(* IEC 61131-3 sources: UniTest/iecUniTest_br/iecUniTest, 121 files *)

(* ---- iecUniTest.typ ---- *)
TYPE
    utTestCase :    STRUCT
        id : UINT; (*Identifier of the test*)
        desc : ARRAY[0..4] OF STRING[255]; (*Description of the test case*)
        state : utTestCaseStates; (*State of the test*)
        msg : STRING[255]; (*Result of the test*)
    END_STRUCT;
    utTestCaseStates :
    (
        ut_SETUP := 0, (**)
        ut_RUNNING := 1, (**)
        ut_PASSED := 2, (**)
        ut_FAILED := 3, (**)
    )
    utTestCaseSummary :    STRUCT
        Id : UINT; (*Id of the test object. Must be unique number*)
        Name : STRING[250]; (*Name of the test object*)
        TotalTests : UINT; (*Total number of tests existing*)
        TestsPassed : UINT; (*Number of tests passed*)
        TestsFailed : UINT; (*Number of tests failed*)
        PassRate : REAL; (*Pass rate % of the tests*)
        TestsRunning : BOOL; (*One or more tests are running*)
        Error : utErrors; (*Error code if error occured*)
    END_STRUCT;
    utErrors :
    (
        ut_NO_ERROR := 0, (**)
        ut_NO_TEST_CASES_DEFINED := 100, (**)
    )
END_TYPE

(* ---- assertArrayEqual_BOOL.st ---- *)
FUNCTION assertArrayEqual_BOOL
    (*https://github.com/tkucic/iecUniTest/blob/main/docs/docs/ns/iecUniTest/fc/assertArrayEqual_BOOL.md*)
    vStop := (size / SIZEOF(act^[0])) - 1;

    FOR i:=0 TO vStop DO
    	pt1 := ADR(act^[i]);
    	pt2 := ADR(xp^[i]);
    	IF pt1^ <> pt2^ THEN
    		assertArrayEqual_BOOL := FALSE;
    		RETURN;
    	END_IF
    END_FOR
    (*If we reach here, all elements are equal*)
    assertArrayEqual_BOOL := TRUE;
    RETURN;

END_FUNCTION

(* ---- assertArrayEqual_BYTE.st ---- *)
FUNCTION assertArrayEqual_BYTE
    (*https://github.com/tkucic/iecUniTest/blob/main/docs/docs/ns/iecUniTest/fc/assertArrayEqual_BYTE.md*)
    vStop := (size / SIZEOF(act[0])) - 1;

    FOR i:=0 TO vStop DO
    	pt1 ACCESS ADR(act[i]);
    	pt2 ACCESS ADR(xp[i]);
    	IF pt1 <> pt2 THEN
    		assertArrayEqual_BYTE := FALSE;
    		RETURN;
    	END_IF
    END_FOR
    (*If we reach here, all elements are equal*)
    assertArrayEqual_BYTE := TRUE;
    RETURN;

END_FUNCTION

(* ---- assertArrayEqual_DATE.st ---- *)
FUNCTION assertArrayEqual_DATE
    (*https://github.com/tkucic/iecUniTest/blob/main/docs/docs/ns/iecUniTest/fc/assertArrayEqual_DATE.md*)
    vStop := (size / SIZEOF(act[0])) - 1;

    FOR i:=0 TO vStop DO
    	pt1 ACCESS ADR(act[i]);
    	pt2 ACCESS ADR(xp[i]);
    	IF pt1 <> pt2 THEN
    		assertArrayEqual_DATE := FALSE;
    		RETURN;
    	END_IF
    END_FOR
    (*If we reach here, all elements are equal*)
    assertArrayEqual_DATE := TRUE;
    RETURN;

END_FUNCTION

(* ---- assertArrayEqual_DATE_AND_TIME.st ---- *)
FUNCTION assertArrayEqual_DATE_AND_TIME
    (*https://github.com/tkucic/iecUniTest/blob/main/docs/docs/ns/iecUniTest/fc/assertArrayEqual_DATE_AND_TIME.md*)
    vStop := (size / SIZEOF(act[0])) - 1;

    FOR i:=0 TO vStop DO
    	pt1 ACCESS ADR(act[i]);
    	pt2 ACCESS ADR(xp[i]);
    	IF pt1 <> pt2 THEN
    		assertArrayEqual_DATE_AND_TIME := FALSE;
    		RETURN;
    	END_IF
    END_FOR
    (*If we reach here, all elements are equal*)
    assertArrayEqual_DATE_AND_TIME := TRUE;
    RETURN;

END_FUNCTION

(* ---- assertArrayEqual_DINT.st ---- *)
FUNCTION assertArrayEqual_DINT
    (*https://github.com/tkucic/iecUniTest/blob/main/docs/docs/ns/iecUniTest/fc/assertArrayEqual_DINT.md*)
    vStop := (size / SIZEOF(act[0])) - 1;

    FOR i:=0 TO vStop DO
    	pt1 ACCESS ADR(act[i]);
    	pt2 ACCESS ADR(xp[i]);
    	IF pt1 <> pt2 THEN
    		assertArrayEqual_DINT := FALSE;
    		RETURN;
    	END_IF
    END_FOR
    (*If we reach here, all elements are equal*)
    assertArrayEqual_DINT := TRUE;
    RETURN;

END_FUNCTION

(* ---- assertArrayEqual_DWORD.st ---- *)
FUNCTION assertArrayEqual_DWORD
    (*https://github.com/tkucic/iecUniTest/blob/main/docs/docs/ns/iecUniTest/fc/assertArrayEqual_DWORD.md*)
    vStop := (size / SIZEOF(act[0])) - 1;

    FOR i:=0 TO vStop DO
    	pt1 ACCESS ADR(act[i]);
    	pt2 ACCESS ADR(xp[i]);
    	IF pt1 <> pt2 THEN
    		assertArrayEqual_DWORD := FALSE;
    		RETURN;
    	END_IF
    END_FOR
    (*If we reach here, all elements are equal*)
    assertArrayEqual_DWORD := TRUE;
    RETURN;

END_FUNCTION

(* ---- assertArrayEqual_INT.st ---- *)
FUNCTION assertArrayEqual_INT
    (*https://github.com/tkucic/iecUniTest/blob/main/docs/docs/ns/iecUniTest/fc/assertArrayEqual_INT.md*)
    vStop := (size / SIZEOF(act[0])) - 1;

    FOR i:=0 TO vStop DO
    	pt1 ACCESS ADR(act[i]);
    	pt2 ACCESS ADR(xp[i]);
    	IF pt1 <> pt2 THEN
    		assertArrayEqual_INT := FALSE;
    		RETURN;
    	END_IF
    END_FOR
    (*If we reach here, all elements are equal*)
    assertArrayEqual_INT := TRUE;
    RETURN;

END_FUNCTION

(* ---- assertArrayEqual_LREAL.st ---- *)
FUNCTION assertArrayEqual_LREAL
    (*https://github.com/tkucic/iecUniTest/blob/main/docs/docs/ns/iecUniTest/fc/assertArrayEqual_LREAL.md*)
    vStop := (size / SIZEOF(act^[0])) - 1;

    FOR i:=0 TO vStop DO
    	pt1 := ADR(act^[i]);
    	pt2 := ADR(xp^[i]);
    	IF pt1^ <> pt2^ THEN
    		assertArrayEqual_LREAL := FALSE;
    		RETURN;
    	END_IF
    END_FOR
    (*If we reach here, all elements are equal*)
    assertArrayEqual_LREAL := TRUE;
    RETURN;

END_FUNCTION

(* ---- assertArrayEqual_REAL.st ---- *)
FUNCTION assertArrayEqual_REAL
    (*https://github.com/tkucic/iecUniTest/blob/main/docs/docs/ns/iecUniTest/fc/assertArrayEqual_REAL.md*)
    vStop := (size / SIZEOF(act^[0])) - 1;

    FOR i:=0 TO vStop DO
    	pt1 := ADR(act^[i]);
    	pt2 := ADR(xp^[i]);
    	IF pt1^ <> pt2^ THEN
    		assertArrayEqual_REAL := FALSE;
    		RETURN;
    	END_IF
    END_FOR
    (*If we reach here, all elements are equal*)
    assertArrayEqual_REAL := TRUE;
    RETURN;

END_FUNCTION

(* ---- assertArrayEqual_SINT.st ---- *)
FUNCTION assertArrayEqual_SINT
    (*https://github.com/tkucic/iecUniTest/blob/main/docs/docs/ns/iecUniTest/fc/assertArrayEqual_SINT.md*)
    vStop := (size / SIZEOF(act[0])) - 1;

    FOR i:=0 TO vStop DO
    	pt1 ACCESS ADR(act[i]);
    	pt2 ACCESS ADR(xp[i]);
    	IF pt1 <> pt2 THEN
    		assertArrayEqual_SINT := FALSE;
    		RETURN;
    	END_IF
    END_FOR
    (*If we reach here, all elements are equal*)
    assertArrayEqual_SINT := TRUE;
    RETURN;

END_FUNCTION

(* ---- assertArrayEqual_STRING.st ---- *)
FUNCTION assertArrayEqual_STRING
    (*https://github.com/tkucic/iecUniTest/blob/main/docs/docs/ns/iecUniTest/fc/assertArrayEqual_STRING.md*)
    vStop := (size / SIZEOF(act[0])) - 1;

    FOR i:=0 TO vStop DO
    	pt1 ACCESS ADR(act[i]);
    	pt2 ACCESS ADR(xp[i]);
    	IF pt1 <> pt2 THEN
    		assertArrayEqual_STRING := FALSE;
    		RETURN;
    	END_IF
    END_FOR
    (*If we reach here, all elements are equal*)
    assertArrayEqual_STRING := TRUE;
    RETURN;

END_FUNCTION

(* ---- assertArrayEqual_TIME.st ---- *)
FUNCTION assertArrayEqual_TIME
    (*https://github.com/tkucic/iecUniTest/blob/main/docs/docs/ns/iecUniTest/fc/assertArrayEqual_TIME.md*)
    vStop := (size / SIZEOF(act^[0])) - 1;

    FOR i:=0 TO vStop DO
    	pt1 := ADR(act^[i]);
    	pt2 := ADR(xp^[i]);
    	IF pt1^ <> pt2^ THEN
    		assertArrayEqual_TIME := FALSE;
    		RETURN;
    	END_IF
    END_FOR
    (*If we reach here, all elements are equal*)
    assertArrayEqual_TIME := TRUE;
    RETURN;

END_FUNCTION

(* ---- assertArrayEqual_TIME_OF_DAY.st ---- *)
FUNCTION assertArrayEqual_TIME_OF_DAY
    (*https://github.com/tkucic/iecUniTest/blob/main/docs/docs/ns/iecUniTest/fc/assertArrayEqual_TIME_OF_DAY.md*)
    vStop := (size / SIZEOF(act^[0])) - 1;

    FOR i:=0 TO vStop DO
    	pt1 := ADR(act^[i]);
    	pt2 := ADR(xp^[i]);
    	IF pt1^ <> pt2^ THEN
    		assertArrayEqual_TIME_OF_DAY := FALSE;
    		RETURN;
    	END_IF
    END_FOR
    (*If we reach here, all elements are equal*)
    assertArrayEqual_TIME_OF_DAY := TRUE;
    RETURN;

END_FUNCTION

(* ---- assertArrayEqual_UDINT.st ---- *)
FUNCTION assertArrayEqual_UDINT
    (*https://github.com/tkucic/iecUniTest/blob/main/docs/docs/ns/iecUniTest/fc/assertArrayEqual_UDINT.md*)
    vStop := (size / SIZEOF(act[0])) - 1;

    FOR i:=0 TO vStop DO
    	pt1 ACCESS ADR(act[i]);
    	pt2 ACCESS ADR(xp[i]);
    	IF pt1 <> pt2 THEN
    		assertArrayEqual_UDINT := FALSE;
    		RETURN;
    	END_IF
    END_FOR
    (*If we reach here, all elements are equal*)
    assertArrayEqual_UDINT := TRUE;
    RETURN;

END_FUNCTION

(* ---- assertArrayEqual_UINT.st ---- *)
FUNCTION assertArrayEqual_UINT
    (*https://github.com/tkucic/iecUniTest/blob/main/docs/docs/ns/iecUniTest/fc/assertArrayEqual_UINT.md*)
    vStop := (size / SIZEOF(act^[0])) - 1;

    FOR i:=0 TO vStop DO
    	pt1 := ADR(act^[i]);
    	pt2 := ADR(xp^[i]);
    	IF pt1^ <> pt2^ THEN
    		assertArrayEqual_UINT := FALSE;
    		RETURN;
    	END_IF
    END_FOR
    (*If we reach here, all elements are equal*)
    assertArrayEqual_UINT := TRUE;
    RETURN;

END_FUNCTION

(* ---- assertArrayEqual_USINT.st ---- *)
FUNCTION assertArrayEqual_USINT
    (*https://github.com/tkucic/iecUniTest/blob/main/docs/docs/ns/iecUniTest/fc/assertArrayEqual_USINT.md*)
    vStop := (size / SIZEOF(act[0])) - 1;

    FOR i:=0 TO vStop DO
    	pt1 ACCESS ADR(act[i]);
    	pt2 ACCESS ADR(xp[i]);
    	IF pt1 <> pt2 THEN
    		assertArrayEqual_USINT := FALSE;
    		RETURN;
    	END_IF
    END_FOR
    (*If we reach here, all elements are equal*)
    assertArrayEqual_USINT := TRUE;
    RETURN;

END_FUNCTION

(* ---- assertArrayEqual_WORD.st ---- *)
FUNCTION assertArrayEqual_WORD
    (*https://github.com/tkucic/iecUniTest/blob/main/docs/docs/ns/iecUniTest/fc/assertArrayEqual_WORD.md*)
    vStop := (size / SIZEOF(act^[0])) - 1;

    FOR i:=0 TO vStop DO
    	pt1 := ADR(act^[i]);
    	pt2 := ADR(xp^[i]);
    	IF pt1^ <> pt2^ THEN
    		assertArrayEqual_WORD := FALSE;
    		RETURN;
    	END_IF
    END_FOR
    (*If we reach here, all elements are equal*)
    assertArrayEqual_WORD := TRUE;
    RETURN;

END_FUNCTION

(* ---- assertArrayEqual_WSTRING.st ---- *)
FUNCTION assertArrayEqual_WSTRING
    (*https://github.com/tkucic/iecUniTest/blob/main/docs/docs/ns/iecUniTest/fc/assertArrayEqual_WSTRING.md*)
    vStop := (size / SIZEOF(act[0])) - 1;

    FOR i:=0 TO vStop DO
    	pt1 ACCESS ADR(act[i]);
    	pt2 ACCESS ADR(xp[i]);
    	IF pt1 <> pt2 THEN
    		assertArrayEqual_WSTRING := FALSE;
    		RETURN;
    	END_IF
    END_FOR
    (*If we reach here, all elements are equal*)
    assertArrayEqual_WSTRING := TRUE;
    RETURN;

END_FUNCTION

(* ---- assertEqual_BOOL.st ---- *)
FUNCTION assertEqual_BOOL
    (*https://github.com/tkucic/iecUniTest/blob/main/docs/docs/ns/iecUniTest/fc/assertEqual_BOOL.md*)
    assertEqual_BOOL := act = xp;
    RETURN;

END_FUNCTION

(* ---- assertEqual_BYTE.st ---- *)
FUNCTION assertEqual_BYTE
    (*https://github.com/tkucic/iecUniTest/blob/main/docs/docs/ns/iecUniTest/fc/assertEqual_BYTE.md*)
    assertEqual_BYTE := act = xp;
    RETURN;

END_FUNCTION

(* ---- assertEqual_DATE.st ---- *)
FUNCTION assertEqual_DATE
    (*https://github.com/tkucic/iecUniTest/blob/main/docs/docs/ns/iecUniTest/fc/assertEqual_DATE.md*)
    assertEqual_DATE := act = xp;
    RETURN;

END_FUNCTION

(* ---- assertEqual_DATE_AND_TIME.st ---- *)
FUNCTION assertEqual_DATE_AND_TIME
    (*https://github.com/tkucic/iecUniTest/blob/main/docs/docs/ns/iecUniTest/fc/assertEqual_DATE_AND_TIME.md*)
    assertEqual_DATE_AND_TIME := act = xp;
    RETURN;

END_FUNCTION

(* ---- assertEqual_DINT.st ---- *)
FUNCTION assertEqual_DINT
    (*https://github.com/tkucic/iecUniTest/blob/main/docs/docs/ns/iecUniTest/fc/assertEqual_DINT.md*)
    assertEqual_DINT := act = xp;
    RETURN;

END_FUNCTION

(* ---- assertEqual_DWORD.st ---- *)
FUNCTION assertEqual_DWORD
    (*https://github.com/tkucic/iecUniTest/blob/main/docs/docs/ns/iecUniTest/fc/assertEqual_DWORD.md*)
    assertEqual_DWORD := act = xp;
    RETURN;

END_FUNCTION

(* ---- assertEqual_INT.st ---- *)
FUNCTION assertEqual_INT
    (*https://github.com/tkucic/iecUniTest/blob/main/docs/docs/ns/iecUniTest/fc/assertEqual_INT.md*)
    assertEqual_INT := act = xp;
    RETURN;

END_FUNCTION

(* ---- assertEqual_LREAL.st ---- *)
FUNCTION assertEqual_LREAL
    (*https://github.com/tkucic/iecUnitTest/blob/main/docs/docs/ns/Global/fc/assertEqual_LREAL.md*)
    assertEqual_LREAL := act = xp;
    RETURN;

END_FUNCTION

(* ---- assertEqual_REAL.st ---- *)
FUNCTION assertEqual_REAL
    (*https://github.com/tkucic/iecUniTest/blob/main/docs/docs/ns/iecUniTest/fc/assertEqual_REAL.md*)
    assertEqual_REAL := act = xp;
    RETURN;

END_FUNCTION

(* ---- assertEqual_SINT.st ---- *)
FUNCTION assertEqual_SINT
    (*https://github.com/tkucic/iecUniTest/blob/main/docs/docs/ns/iecUniTest/fc/assertEqual_SINT.md*)
    assertEqual_SINT := act = xp;
    RETURN;

END_FUNCTION

(* ---- assertEqual_STRING.st ---- *)
FUNCTION assertEqual_STRING
    (*https://github.com/tkucic/iecUniTest/blob/main/docs/docs/ns/iecUniTest/fc/assertEqual_STRING.md*)
    assertEqual_STRING := act = xp;
    RETURN;

END_FUNCTION

(* ---- assertEqual_TIME.st ---- *)
FUNCTION assertEqual_TIME
    (*https://github.com/tkucic/iecUniTest/blob/main/docs/docs/ns/iecUniTest/fc/assertEqual_TIME.md*)
    assertEqual_TIME := act = xp;
    RETURN;

END_FUNCTION

(* ---- assertEqual_TIME_OF_DAY.st ---- *)
FUNCTION assertEqual_TIME_OF_DAY
    (*https://github.com/tkucic/iecUnitTest/blob/main/docs/docs/ns/Global/fc/assertEqual_TIME_OF_DAY.md*)
    assertEqual_TIME_OF_DAY := act = xp;
    RETURN;

END_FUNCTION

(* ---- assertEqual_UDINT.st ---- *)
FUNCTION assertEqual_UDINT
    (*https://github.com/tkucic/iecUniTest/blob/main/docs/docs/ns/iecUniTest/fc/assertEqual_UDINT.md*)
    assertEqual_UDINT := act = xp;
    RETURN;

END_FUNCTION

(* ---- assertEqual_UINT.st ---- *)
FUNCTION assertEqual_UINT
    (*https://github.com/tkucic/iecUniTest/blob/main/docs/docs/ns/iecUniTest/fc/assertEqual_UINT.md*)
    assertEqual_UINT := act = xp;
    RETURN;

END_FUNCTION

(* ---- assertEqual_USINT.st ---- *)
FUNCTION assertEqual_USINT
    (*https://github.com/tkucic/iecUniTest/blob/main/docs/docs/ns/iecUniTest/fc/assertEqual_USINT.md*)
    assertEqual_USINT := act = xp;
    RETURN;

END_FUNCTION

(* ---- assertEqual_WORD.st ---- *)
FUNCTION assertEqual_WORD
    (*https://github.com/tkucic/iecUnitTest/blob/main/docs/docs/ns/Global/fc/assertEqual_WORD.md*)
    assertEqual_WORD := act = xp;
    RETURN;

END_FUNCTION

(* ---- assertEqual_WSTRING.st ---- *)
FUNCTION assertEqual_WSTRING
    (*https://github.com/tkucic/iecUniTest/blob/main/docs/docs/ns/iecUniTest/fc/assertEqual_WSTRING.md*)
    assertEqual_WSTRING := act = xp;
    RETURN;

END_FUNCTION

(* ---- assertFalse.st ---- *)
FUNCTION assertFalse
    (*https://github.com/tkucic/iecUniTest/blob/main/docs/docs/ns/iecUniTest/fc/assertFalse.md*)
    assertFalse := NOT condition;
    RETURN;

END_FUNCTION

(* ---- assertGreater_BYTE.st ---- *)
FUNCTION assertGreater_BYTE
    (*https://github.com/tkucic/iecUniTest/blob/main/docs/docs/ns/iecUniTest/fc/assertGreater_BYTE.md*)
    assertGreater_BYTE := act > xp;
    RETURN;

END_FUNCTION

(* ---- assertGreater_DATE.st ---- *)
FUNCTION assertGreater_DATE
    (*https://github.com/tkucic/iecUniTest/blob/main/docs/docs/ns/iecUniTest/fc/assertGreater_DATE.md*)
    assertGreater_DATE := act > xp;
    RETURN;

END_FUNCTION

(* ---- assertGreater_DATE_AND_TIME.st ---- *)
FUNCTION assertGreater_DATE_AND_TIME
    (*https://github.com/tkucic/iecUniTest/blob/main/docs/docs/ns/iecUniTest/fc/assertGreater_DATE_AND_TIME.md*)
    assertGreater_DATE_AND_TIME := act > xp;
    RETURN;

END_FUNCTION

(* ---- assertGreater_DINT.st ---- *)
FUNCTION assertGreater_DINT
    (*https://github.com/tkucic/iecUniTest/blob/main/docs/docs/ns/iecUniTest/fc/assertGreater_DINT.md*)
    assertGreater_DINT := act > xp;
    RETURN;

END_FUNCTION

(* ---- assertGreater_DWORD.st ---- *)
FUNCTION assertGreater_DWORD
    (*https://github.com/tkucic/iecUniTest/blob/main/docs/docs/ns/iecUniTest/fc/assertGreater_DWORD.md*)
    assertGreater_DWORD := act > xp;
    RETURN;

END_FUNCTION

(* ---- assertGreater_INT.st ---- *)
FUNCTION assertGreater_INT
    (*https://github.com/tkucic/iecUniTest/blob/main/docs/docs/ns/iecUniTest/fc/assertGreater_INT.md*)
    assertGreater_INT := act > xp;
    RETURN;

END_FUNCTION

(* ---- assertGreater_LREAL.st ---- *)
FUNCTION assertGreater_LREAL
    (*https://github.com/tkucic/iecUniTest/blob/main/docs/docs/ns/iecUniTest/fc/assertGreater_LREAL.md*)
    assertGreater_LREAL := act > xp;
    RETURN;

END_FUNCTION

(* ---- assertGreater_REAL.st ---- *)
FUNCTION assertGreater_REAL
    (*https://github.com/tkucic/iecUniTest/blob/main/docs/docs/ns/iecUniTest/fc/assertGreater_REAL.md*)
    assertGreater_REAL := act > xp;
    RETURN;

END_FUNCTION

(* ---- assertGreater_SINT.st ---- *)
FUNCTION assertGreater_SINT
    (*https://github.com/tkucic/iecUniTest/blob/main/docs/docs/ns/iecUniTest/fc/assertGreater_SINT.md*)
    assertGreater_SINT := act > xp;
    RETURN;

END_FUNCTION

(* ---- assertGreater_TIME.st ---- *)
FUNCTION assertGreater_TIME
    (*https://github.com/tkucic/iecUniTest/blob/main/docs/docs/ns/iecUniTest/fc/assertGreater_TIME.md*)
    assertGreater_TIME := act > xp;
    RETURN;

END_FUNCTION

(* ---- assertGreater_TIME_OF_DAY.st ---- *)
FUNCTION assertGreater_TIME_OF_DAY
    (*https://github.com/tkucic/iecUniTest/blob/main/docs/docs/ns/iecUniTest/fc/assertGreater_TIME_OF_DAY.md*)
    assertGreater_TIME_OF_DAY := act > xp;
    RETURN;

END_FUNCTION

(* ---- assertGreater_UDINT.st ---- *)
FUNCTION assertGreater_UDINT
    (*https://github.com/tkucic/iecUniTest/blob/main/docs/docs/ns/iecUniTest/fc/assertGreater_UDINT.md*)
    assertGreater_UDINT := act > xp;
    RETURN;

END_FUNCTION

(* ---- assertGreater_UINT.st ---- *)
FUNCTION assertGreater_UINT
    (*https://github.com/tkucic/iecUniTest/blob/main/docs/docs/ns/iecUniTest/fc/assertGreater_UINT.md*)
    assertGreater_UINT := act > xp;
    RETURN;

END_FUNCTION

(* ---- assertGreater_USINT.st ---- *)
FUNCTION assertGreater_USINT
    (*https://github.com/tkucic/iecUniTest/blob/main/docs/docs/ns/iecUniTest/fc/assertGreater_USINT.md*)
    assertGreater_USINT := act > xp;
    RETURN;

END_FUNCTION

(* ---- assertGreater_WORD.st ---- *)
FUNCTION assertGreater_WORD
    (*https://github.com/tkucic/iecUniTest/blob/main/docs/docs/ns/iecUniTest/fc/assertGreater_WORD.md*)
    assertGreater_WORD := act > xp;
    RETURN;

END_FUNCTION

(* ---- assertGreaterEqual_BYTE.st ---- *)
FUNCTION assertGreaterEqual_BYTE
    (*https://github.com/tkucic/iecUniTest/blob/main/docs/docs/ns/iecUniTest/fc/assertGreaterEqual_BYTE.md*)
    assertGreaterEqual_BYTE := act >= xp;
    RETURN;

END_FUNCTION

(* ---- assertGreaterEqual_DATE.st ---- *)
FUNCTION assertGreaterEqual_DATE
    (*https://github.com/tkucic/iecUniTest/blob/main/docs/docs/ns/iecUniTest/fc/assertGreaterEqual_DATE.md*)
    assertGreaterEqual_DATE := act >= xp;
    RETURN;

END_FUNCTION

(* ---- assertGreaterEqual_DATE_AND_TIME.st ---- *)
FUNCTION assertGreaterEqual_DATE_AND_TIME
    (*https://github.com/tkucic/iecUniTest/blob/main/docs/docs/ns/iecUniTest/fc/assertGreaterEqual_DATE_AND_TIME.md*)
    assertGreaterEqual_DATE_AND_TIME := act >= xp;
    RETURN;

END_FUNCTION

(* ---- assertGreaterEqual_DINT.st ---- *)
FUNCTION assertGreaterEqual_DINT
    (*https://github.com/tkucic/iecUnitTest/blob/main/docs/docs/ns/Global/fc/assertGreaterEqual_DINT.md*)
    assertGreaterEqual_DINT := act >= xp;
    RETURN;

END_FUNCTION

(* ---- assertGreaterEqual_DWORD.st ---- *)
FUNCTION assertGreaterEqual_DWORD
    (*https://github.com/tkucic/iecUniTest/blob/main/docs/docs/ns/iecUniTest/fc/assertGreaterEqual_DWORD.md*)
    assertGreaterEqual_DWORD := act >= xp;
    RETURN;

END_FUNCTION

(* ---- assertGreaterEqual_INT.st ---- *)
FUNCTION assertGreaterEqual_INT
    (*https://github.com/tkucic/iecUnitTest/blob/main/docs/docs/ns/Global/fc/assertGreaterEqual_INT.md*)
    assertGreaterEqual_INT := act >= xp;
    RETURN;

END_FUNCTION

(* ---- assertGreaterEqual_LREAL.st ---- *)
FUNCTION assertGreaterEqual_LREAL
    (*https://github.com/tkucic/iecUnitTest/blob/main/docs/docs/ns/Global/fc/assertGreaterEqual_LREAL.md*)
    assertGreaterEqual_LREAL := act >= xp;
    RETURN;

END_FUNCTION

(* ---- assertGreaterEqual_REAL.st ---- *)
FUNCTION assertGreaterEqual_REAL
    (*https://github.com/tkucic/iecUniTest/blob/main/docs/docs/ns/iecUniTest/fc/assertGreaterEqual_REAL.md*)
    assertGreaterEqual_REAL := act >= xp;
    RETURN;

END_FUNCTION

(* ---- assertGreaterEqual_SINT.st ---- *)
FUNCTION assertGreaterEqual_SINT
    (*https://github.com/tkucic/iecUniTest/blob/main/docs/docs/ns/iecUniTest/fc/assertGreaterEqual_SINT.md*)
    assertGreaterEqual_SINT := act >= xp;
    RETURN;

END_FUNCTION

(* ---- assertGreaterEqual_TIME.st ---- *)
FUNCTION assertGreaterEqual_TIME
    (*https://github.com/tkucic/iecUniTest/blob/main/docs/docs/ns/iecUniTest/fc/assertGreaterEqual_TIME.md*)
    assertGreaterEqual_TIME := act >= xp;
    RETURN;

END_FUNCTION

(* ---- assertGreaterEqual_TIME_OF_DAY.st ---- *)
FUNCTION assertGreaterEqual_TIME_OF_DAY
    (*https://github.com/tkucic/iecUniTest/blob/main/docs/docs/ns/iecUniTest/fc/assertGreaterEqual_TIME_OF_DAY.md*)
    assertGreaterEqual_TIME_OF_DAY := act >= xp;
    RETURN;

END_FUNCTION

(* ---- assertGreaterEqual_UDINT.st ---- *)
FUNCTION assertGreaterEqual_UDINT
    (*https://github.com/tkucic/iecUniTest/blob/main/docs/docs/ns/iecUniTest/fc/assertGreaterEqual_UDINT.md*)
    assertGreaterEqual_UDINT := act >= xp;
    RETURN;

END_FUNCTION

(* ---- assertGreaterEqual_UINT.st ---- *)
FUNCTION assertGreaterEqual_UINT
    (*https://github.com/tkucic/iecUniTest/blob/main/docs/docs/ns/iecUniTest/fc/assertGreaterEqual_UINT.md*)
    assertGreaterEqual_UINT := act >= xp;
    RETURN;

END_FUNCTION

(* ---- assertGreaterEqual_USINT.st ---- *)
FUNCTION assertGreaterEqual_USINT
    (*https://github.com/tkucic/iecUniTest/blob/main/docs/docs/ns/iecUniTest/fc/assertGreaterEqual_USINT.md*)
    assertGreaterEqual_USINT := act >= xp;
    RETURN;

END_FUNCTION

(* ---- assertGreaterEqual_WORD.st ---- *)
FUNCTION assertGreaterEqual_WORD
    (*https://github.com/tkucic/iecUniTest/blob/main/docs/docs/ns/iecUniTest/fc/assertGreaterEqual_WORD.md*)
    assertGreaterEqual_WORD := act >= xp;
    RETURN;

END_FUNCTION

(* ---- assertLess_BYTE.st ---- *)
FUNCTION assertLess_BYTE
    (*https://github.com/tkucic/iecUniTest/blob/main/docs/docs/ns/iecUniTest/fc/assertLess_BYTE.md*)
    assertLess_BYTE := act < xp;
    RETURN;

END_FUNCTION

(* ---- assertLess_DATE.st ---- *)
FUNCTION assertLess_DATE
    (*https://github.com/tkucic/iecUnitTest/blob/main/docs/docs/ns/Global/fc/assertLess_DATE.md*)
    assertLess_DATE := act < xp;
    RETURN;

END_FUNCTION

(* ---- assertLess_DATE_AND_TIME.st ---- *)
FUNCTION assertLess_DATE_AND_TIME
    (*https://github.com/tkucic/iecUniTest/blob/main/docs/docs/ns/iecUniTest/fc/assertLess_DATE_AND_TIME.md*)
    assertLess_DATE_AND_TIME := act < xp;
    RETURN;

END_FUNCTION

(* ---- assertLess_DINT.st ---- *)
FUNCTION assertLess_DINT
    (*https://github.com/tkucic/iecUniTest/blob/main/docs/docs/ns/iecUniTest/fc/assertLess_DINT.md*)
    assertLess_DINT := act < xp;
    RETURN;

END_FUNCTION

(* ---- assertLess_DWORD.st ---- *)
FUNCTION assertLess_DWORD
    (*https://github.com/tkucic/iecUniTest/blob/main/docs/docs/ns/iecUniTest/fc/assertLess_DWORD.md*)
    assertLess_DWORD := act < xp;
    RETURN;

END_FUNCTION

(* ---- assertLess_INT.st ---- *)
FUNCTION assertLess_INT
    (*https://github.com/tkucic/iecUniTest/blob/main/docs/docs/ns/iecUniTest/fc/assertLess_INT.md*)
    assertLess_INT := act < xp;
    RETURN;

END_FUNCTION

(* ---- assertLess_LREAL.st ---- *)
FUNCTION assertLess_LREAL
    (*https://github.com/tkucic/iecUniTest/blob/main/docs/docs/ns/iecUniTest/fc/assertLess_LREAL.md*)
    assertLess_LREAL := act < xp;
    RETURN;

END_FUNCTION

(* ---- assertLess_REAL.st ---- *)
FUNCTION assertLess_REAL
    (*https://github.com/tkucic/iecUniTest/blob/main/docs/docs/ns/iecUniTest/fc/assertLess_REAL.md*)
    assertLess_REAL := act < xp;
    RETURN;

END_FUNCTION

(* ---- assertLess_SINT.st ---- *)
FUNCTION assertLess_SINT
    (*https://github.com/tkucic/iecUniTest/blob/main/docs/docs/ns/iecUniTest/fc/assertLess_SINT.md*)
    assertLess_SINT := act < xp;
    RETURN;

END_FUNCTION

(* ---- assertLess_TIME.st ---- *)
FUNCTION assertLess_TIME
    (*https://github.com/tkucic/iecUniTest/blob/main/docs/docs/ns/iecUniTest/fc/assertLess_TIME.md*)
    assertLess_TIME := act < xp;
    RETURN;

END_FUNCTION

(* ---- assertLess_TIME_OF_DAY.st ---- *)
FUNCTION assertLess_TIME_OF_DAY
    (*https://github.com/tkucic/iecUniTest/blob/main/docs/docs/ns/iecUniTest/fc/assertLess_TIME_OF_DAY.md*)
    assertLess_TIME_OF_DAY := act < xp;
    RETURN;

END_FUNCTION

(* ---- assertLess_UDINT.st ---- *)
FUNCTION assertLess_UDINT
    (*https://github.com/tkucic/iecUniTest/blob/main/docs/docs/ns/iecUniTest/fc/assertLess_UDINT.md*)
    assertLess_UDINT := act < xp;
    RETURN;

END_FUNCTION

(* ---- assertLess_UINT.st ---- *)
FUNCTION assertLess_UINT
    (*https://github.com/tkucic/iecUnitTest/blob/main/docs/docs/ns/Global/fc/assertLess_UINT.md*)
    assertLess_UINT := act < xp;
    RETURN;

END_FUNCTION

(* ---- assertLess_USINT.st ---- *)
FUNCTION assertLess_USINT
    (*https://github.com/tkucic/iecUniTest/blob/main/docs/docs/ns/iecUniTest/fc/assertLess_USINT.md*)
    assertLess_USINT := act < xp;
    RETURN;

END_FUNCTION

(* ---- assertLess_WORD.st ---- *)
FUNCTION assertLess_WORD
    (*https://github.com/tkucic/iecUniTest/blob/main/docs/docs/ns/iecUniTest/fc/assertLess_WORD.md*)
    assertLess_WORD := act < xp;
    RETURN;

END_FUNCTION

(* ---- assertLessEqual_BYTE.st ---- *)
FUNCTION assertLessEqual_BYTE
    (*https://github.com/tkucic/iecUniTest/blob/main/docs/docs/ns/iecUniTest/fc/assertLessEqual_BYTE.md*)
    assertLessEqual_BYTE := act <= xp;
    RETURN;

END_FUNCTION

(* ---- assertLessEqual_DATE.st ---- *)
FUNCTION assertLessEqual_DATE
    (*https://github.com/tkucic/iecUniTest/blob/main/docs/docs/ns/iecUniTest/fc/assertLessEqual_DATE.md*)
    assertLessEqual_DATE := act <= xp;
    RETURN;

END_FUNCTION

(* ---- assertLessEqual_DATE_AND_TIME.st ---- *)
FUNCTION assertLessEqual_DATE_AND_TIME
    (*https://github.com/tkucic/iecUniTest/blob/main/docs/docs/ns/iecUniTest/fc/assertLessEqual_DATE_AND_TIME.md*)
    assertLessEqual_DATE_AND_TIME := act <= xp;
    RETURN;

END_FUNCTION

(* ---- assertLessEqual_DINT.st ---- *)
FUNCTION assertLessEqual_DINT
    (*https://github.com/tkucic/iecUniTest/blob/main/docs/docs/ns/iecUniTest/fc/assertLessEqual_DINT.md*)
    assertLessEqual_DINT := act <= xp;
    RETURN;

END_FUNCTION

(* ---- assertLessEqual_DWORD.st ---- *)
FUNCTION assertLessEqual_DWORD
    (*https://github.com/tkucic/iecUniTest/blob/main/docs/docs/ns/iecUniTest/fc/assertLessEqual_DWORD.md*)
    assertLessEqual_DWORD := act <= xp;
    RETURN;

END_FUNCTION

(* ---- assertLessEqual_INT.st ---- *)
FUNCTION assertLessEqual_INT
    (*https://github.com/tkucic/iecUniTest/blob/main/docs/docs/ns/iecUniTest/fc/assertLessEqual_INT.md*)
    assertLessEqual_INT := act <= xp;
    RETURN;

END_FUNCTION

(* ---- assertLessEqual_LREAL.st ---- *)
FUNCTION assertLessEqual_LREAL
    (*https://github.com/tkucic/iecUniTest/blob/main/docs/docs/ns/iecUniTest/fc/assertLessEqual_LREAL.md*)
    assertLessEqual_LREAL := act <= xp;
    RETURN;

END_FUNCTION

(* ---- assertLessEqual_REAL.st ---- *)
FUNCTION assertLessEqual_REAL
    (*https://github.com/tkucic/iecUniTest/blob/main/docs/docs/ns/iecUniTest/fc/assertLessEqual_REAL.md*)
    assertLessEqual_REAL := act <= xp;
    RETURN;

END_FUNCTION

(* ---- assertLessEqual_SINT.st ---- *)
FUNCTION assertLessEqual_SINT
    (*https://github.com/tkucic/iecUniTest/blob/main/docs/docs/ns/iecUniTest/fc/assertLessEqual_SINT.md*)
    assertLessEqual_SINT := act <= xp;
    RETURN;

END_FUNCTION

(* ---- assertLessEqual_TIME.st ---- *)
FUNCTION assertLessEqual_TIME
    (*https://github.com/tkucic/iecUniTest/blob/main/docs/docs/ns/iecUniTest/fc/assertLessEqual_TIME.md*)
    assertLessEqual_TIME := act <= xp;
    RETURN;

END_FUNCTION

(* ---- assertLessEqual_TIME_OF_DAY.st ---- *)
FUNCTION assertLessEqual_TIME_OF_DAY
    (*https://github.com/tkucic/iecUniTest/blob/main/docs/docs/ns/iecUniTest/fc/assertLessEqual_TIME_OF_DAY.md*)
    assertLessEqual_TIME_OF_DAY := act <= xp;
    RETURN;

END_FUNCTION

(* ---- assertLessEqual_UDINT.st ---- *)
FUNCTION assertLessEqual_UDINT
    (*https://github.com/tkucic/iecUniTest/blob/main/docs/docs/ns/iecUniTest/fc/assertLessEqual_UDINT.md*)
    assertLessEqual_UDINT := act <= xp;
    RETURN;

END_FUNCTION

(* ---- assertLessEqual_UINT.st ---- *)
FUNCTION assertLessEqual_UINT
    (*https://github.com/tkucic/iecUniTest/blob/main/docs/docs/ns/iecUniTest/fc/assertLessEqual_UINT.md*)
    assertLessEqual_UINT := act <= xp;
    RETURN;

END_FUNCTION

(* ---- assertLessEqual_USINT.st ---- *)
FUNCTION assertLessEqual_USINT
    (*https://github.com/tkucic/iecUniTest/blob/main/docs/docs/ns/iecUniTest/fc/assertLessEqual_USINT.md*)
    assertLessEqual_USINT := act <= xp;
    RETURN;

END_FUNCTION

(* ---- assertLessEqual_WORD.st ---- *)
FUNCTION assertLessEqual_WORD
    (*https://github.com/tkucic/iecUniTest/blob/main/docs/docs/ns/iecUniTest/fc/assertLessEqual_WORD.md*)
    assertLessEqual_WORD := act <= xp;
    RETURN;

END_FUNCTION

(* ---- assertNotEqual_BOOL.st ---- *)
FUNCTION assertNotEqual_BOOL
    (*https://github.com/tkucic/iecUniTest/blob/main/docs/docs/ns/iecUniTest/fc/assertNotEqual_BOOL.md*)
    assertNotEqual_BOOL := act <> xp;
    RETURN;

END_FUNCTION

(* ---- assertNotEqual_BYTE.st ---- *)
FUNCTION assertNotEqual_BYTE
    (*https://github.com/tkucic/iecUniTest/blob/main/docs/docs/ns/iecUniTest/fc/assertNotEqual_BYTE.md*)
    assertNotEqual_BYTE := act <> xp;
    RETURN;

END_FUNCTION

(* ---- assertNotEqual_DATE.st ---- *)
FUNCTION assertNotEqual_DATE
    (*https://github.com/tkucic/iecUniTest/blob/main/docs/docs/ns/iecUniTest/fc/assertNotEqual_DATE.md*)
    assertNotEqual_DATE := act <> xp;
    RETURN;

END_FUNCTION

(* ---- assertNotEqual_DATE_AND_TIME.st ---- *)
FUNCTION assertNotEqual_DATE_AND_TIME
    (*https://github.com/tkucic/iecUnitTest/blob/main/docs/docs/ns/Global/fc/assertNotEqual_DATE_AND_TIME.md*)
    assertNotEqual_DATE_AND_TIME := act <> xp;
    RETURN;

END_FUNCTION

(* ---- assertNotEqual_DINT.st ---- *)
FUNCTION assertNotEqual_DINT
    (*https://github.com/tkucic/iecUniTest/blob/main/docs/docs/ns/iecUniTest/fc/assertNotEqual_DINT.md*)
    assertNotEqual_DINT := act <> xp;
    RETURN;

END_FUNCTION

(* ---- assertNotEqual_DWORD.st ---- *)
FUNCTION assertNotEqual_DWORD
    (*https://github.com/tkucic/iecUniTest/blob/main/docs/docs/ns/iecUniTest/fc/assertNotEqual_DWORD.md*)
    assertNotEqual_DWORD := act <> xp;
    RETURN;

END_FUNCTION

(* ---- assertNotEqual_INT.st ---- *)
FUNCTION assertNotEqual_INT
    (*https://github.com/tkucic/iecUniTest/blob/main/docs/docs/ns/iecUniTest/fc/assertNotEqual_INT.md*)
    assertNotEqual_INT := act <> xp;
    RETURN;

END_FUNCTION

(* ---- assertNotEqual_LREAL.st ---- *)
FUNCTION assertNotEqual_LREAL
    (*https://github.com/tkucic/iecUniTest/blob/main/docs/docs/ns/iecUniTest/fc/assertNotEqual_LREAL.md*)
    assertNotEqual_LREAL := act <> xp;
    RETURN;

END_FUNCTION

(* ---- assertNotEqual_REAL.st ---- *)
FUNCTION assertNotEqual_REAL
    (*https://github.com/tkucic/iecUniTest/blob/main/docs/docs/ns/iecUniTest/fc/assertNotEqual_REAL.md*)
    assertNotEqual_REAL := act <> xp;
    RETURN;

END_FUNCTION

(* ---- assertNotEqual_SINT.st ---- *)
FUNCTION assertNotEqual_SINT
    (*https://github.com/tkucic/iecUniTest/blob/main/docs/docs/ns/iecUniTest/fc/assertNotEqual_SINT.md*)
    assertNotEqual_SINT := act <> xp;
    RETURN;

END_FUNCTION

(* ---- assertNotEqual_STRING.st ---- *)
FUNCTION assertNotEqual_STRING
    (*https://github.com/tkucic/iecUniTest/blob/main/docs/docs/ns/iecUniTest/fc/assertNotEqual_STRING.md*)
    assertNotEqual_STRING := act <> xp;
    RETURN;

END_FUNCTION

(* ---- assertNotEqual_TIME.st ---- *)
FUNCTION assertNotEqual_TIME
    (*https://github.com/tkucic/iecUniTest/blob/main/docs/docs/ns/iecUniTest/fc/assertNotEqual_TIME.md*)
    assertNotEqual_TIME := act <> xp;
    RETURN;

END_FUNCTION

(* ---- assertNotEqual_TIME_OF_DAY.st ---- *)
FUNCTION assertNotEqual_TIME_OF_DAY
    (*https://github.com/tkucic/iecUnitTest/blob/main/docs/docs/ns/Global/fc/assertNotEqual_TIME_OF_DAY.md*)
    assertNotEqual_TIME_OF_DAY := act <> xp;
    RETURN;

END_FUNCTION

(* ---- assertNotEqual_UDINT.st ---- *)
FUNCTION assertNotEqual_UDINT
    (*https://github.com/tkucic/iecUniTest/blob/main/docs/docs/ns/iecUniTest/fc/assertNotEqual_UDINT.md*)
    assertNotEqual_UDINT := act <> xp;
    RETURN;

END_FUNCTION

(* ---- assertNotEqual_UINT.st ---- *)
FUNCTION assertNotEqual_UINT
    (*https://github.com/tkucic/iecUniTest/blob/main/docs/docs/ns/iecUniTest/fc/assertNotEqual_UINT.md*)
    assertNotEqual_UINT := act <> xp;
    RETURN;

END_FUNCTION

(* ---- assertNotEqual_USINT.st ---- *)
FUNCTION assertNotEqual_USINT
    (*https://github.com/tkucic/iecUnitTest/blob/main/docs/docs/ns/Global/fc/assertNotEqual_USINT.md*)
    assertNotEqual_USINT := act <> xp;
    RETURN;

END_FUNCTION

(* ---- assertNotEqual_WORD.st ---- *)
FUNCTION assertNotEqual_WORD
    (*https://github.com/tkucic/iecUniTest/blob/main/docs/docs/ns/iecUniTest/fc/assertNotEqual_WORD.md*)
    assertNotEqual_WORD := act <> xp;
    RETURN;

END_FUNCTION

(* ---- assertNotEqual_WSTRING.st ---- *)
FUNCTION assertNotEqual_WSTRING
    (*https://github.com/tkucic/iecUniTest/blob/main/docs/docs/ns/iecUniTest/fc/assertNotEqual_WSTRING.md*)
    assertNotEqual_WSTRING := act <> xp;
    RETURN;

END_FUNCTION

(* ---- assertTrue.st ---- *)
FUNCTION assertTrue
    (*https://github.com/tkucic/iecUniTest/blob/main/docs/docs/ns/iecUniTest/fc/assertTrue.md*)
    assertTrue := condition;
    RETURN;

END_FUNCTION

(* ---- iecUniTest.fun ---- *)
FUNCTION_BLOCK utTestSuite (* Enables running, resetting and reporting for tests cases defined of a POU under test *)(* https://github.com/tkucic/iecUniTest/blob/main/docs/docs/ns/iecUniTest/fb/utTestSuite.md *)
    VAR_INPUT
        Id : UINT; (*Id of the test object. Must be unique number*)
        Name : STRING[250]; (*Name of the test object*)
        RunTests : BOOL; (*Starts all tests that are in setup state. Sets state to running.*)
        ResetTests : BOOL; (*Sets state to setup on test cases that are ut_PASSED or ut_FAILED.*)
    END_VAR
    VAR_IN_OUT
        TestCases : ARRAY[0..20] OF utTestCase; (*Array of test case definition*)
    END_VAR
    VAR_OUTPUT
        Summary : utTestCaseSummary; (*Summary of the test results*)
    END_VAR
    VAR
        i : UINT; (*Iterator variable*)
        runCmd : R_TRIG; (*Trigger to prevent constant run commands*)
        resetCmd : R_TRIG; (*Trigger to prevent constant reset commands*)
    END_VAR
END_FUNCTION_BLOCK
FUNCTION_BLOCK utTestReporter (* Provides feedback on the status of tests on a system scale *)(* https://github.com/tkucic/iecUniTest/blob/main/docs/docs/ns/iecUniTest/fb/utTestReporter.md *)
    VAR_IN_OUT
        Results : ARRAY[0..500] OF utTestCaseSummary; (*Summaries of tests for each POU under test*)
    END_VAR
    VAR_OUTPUT
        NrPousUnderTest : UINT; (*Total number of POUs under test*)
        NrOfTests : UINT; (*Total number of tests*)
        NrTestsPassed : UINT; (*Number of tests passed*)
        NrTestsFailed : UINT; (*Number of tests failed*)
        PassRate : REAL; (*Total pass rate*)
        TestsInProgress : BOOL; (*Indicates that one or more tests are in progress*)
        Error : BOOL; (*Indicates that one or more tests are in error state*)
    END_VAR
    VAR
        i : UINT; (*Iterator variable*)
    END_VAR
END_FUNCTION_BLOCK
FUNCTION assertFalse : BOOL (* Returns TRUE if condition is NOT TRUE *)(* https://github.com/tkucic/iecUniTest/blob/main/docs/docs/ns/iecUniTest/fc/assertFalse.md *)
    VAR_INPUT
        condition : BOOL; (*Variable to test*)
    END_VAR
END_FUNCTION
FUNCTION assertEqual_BOOL : BOOL (* Returns TRUE if act = xp. *)(* https://github.com/tkucic/iecUniTest/blob/main/docs/docs/ns/iecUniTest/fc/assertEqual_BOOL.md *)
    VAR_INPUT
        act : BOOL; (*Variable to test*)
        xp : BOOL; (*Variable to test against*)
    END_VAR
END_FUNCTION
FUNCTION assertEqual_BYTE : BOOL (* Returns TRUE if act = xp. *)(* https://github.com/tkucic/iecUniTest/blob/main/docs/docs/ns/iecUniTest/fc/assertEqual_BYTE.md *)
    VAR_INPUT
        act : BYTE; (*Variable to test*)
        xp : BYTE; (*Variable to test against*)
    END_VAR
END_FUNCTION
FUNCTION assertEqual_WORD : BOOL (* Returns TRUE if act = xp. *)(* https://github.com/tkucic/iecUniTest/blob/main/docs/docs/ns/iecUniTest/fc/assertEqual_WORD.md *)
    VAR_INPUT
        act : WORD; (*Variable to test*)
        xp : WORD; (*Variable to test against*)
    END_VAR
END_FUNCTION
FUNCTION assertEqual_DWORD : BOOL (* Returns TRUE if act = xp. *)(* https://github.com/tkucic/iecUniTest/blob/main/docs/docs/ns/iecUniTest/fc/assertEqual_DWORD.md *)
    VAR_INPUT
        act : DWORD; (*Variable to test*)
        xp : DWORD; (*Variable to test against*)
    END_VAR
END_FUNCTION
FUNCTION assertEqual_SINT : BOOL (* Returns TRUE if act = xp. *)(* https://github.com/tkucic/iecUniTest/blob/main/docs/docs/ns/iecUniTest/fc/assertEqual_SINT.md *)
    VAR_INPUT
        act : SINT; (*Variable to test*)
        xp : SINT; (*Variable to test against*)
    END_VAR
END_FUNCTION
FUNCTION assertEqual_USINT : BOOL (* Returns TRUE if act = xp. *)(* https://github.com/tkucic/iecUniTest/blob/main/docs/docs/ns/iecUniTest/fc/assertEqual_USINT.md *)
    VAR_INPUT
        act : USINT; (*Variable to test*)
        xp : USINT; (*Variable to test against*)
    END_VAR
END_FUNCTION
FUNCTION assertEqual_INT : BOOL (* Returns TRUE if act = xp. *)(* https://github.com/tkucic/iecUniTest/blob/main/docs/docs/ns/iecUniTest/fc/assertEqual_INT.md *)
    VAR_INPUT
        act : INT; (*Variable to test*)
        xp : INT; (*Variable to test against*)
    END_VAR
END_FUNCTION
FUNCTION assertEqual_UINT : BOOL (* Returns TRUE if act = xp. *)(* https://github.com/tkucic/iecUniTest/blob/main/docs/docs/ns/iecUniTest/fc/assertEqual_UINT.md *)
    VAR_INPUT
        act : UINT; (*Variable to test*)
        xp : UINT; (*Variable to test against*)
    END_VAR
END_FUNCTION
FUNCTION assertEqual_DINT : BOOL (* Returns TRUE if act = xp. *)(* https://github.com/tkucic/iecUniTest/blob/main/docs/docs/ns/iecUniTest/fc/assertEqual_DINT.md *)
    VAR_INPUT
        act : DINT; (*Variable to test*)
        xp : DINT; (*Variable to test against*)
    END_VAR
END_FUNCTION
FUNCTION assertEqual_UDINT : BOOL (* Returns TRUE if act = xp. *)(* https://github.com/tkucic/iecUniTest/blob/main/docs/docs/ns/iecUniTest/fc/assertEqual_UDINT.md *)
    VAR_INPUT
        act : UDINT; (*Variable to test*)
        xp : UDINT; (*Variable to test against*)
    END_VAR
END_FUNCTION
FUNCTION assertEqual_REAL : BOOL (* Returns TRUE if act = xp. *)(* https://github.com/tkucic/iecUniTest/blob/main/docs/docs/ns/iecUniTest/fc/assertEqual_REAL.md *)
    VAR_INPUT
        act : REAL; (*Variable to test*)
        xp : REAL; (*Variable to test against*)
    END_VAR
END_FUNCTION
FUNCTION assertEqual_LREAL : BOOL (* Returns TRUE if act = xp. *)(* https://github.com/tkucic/iecUniTest/blob/main/docs/docs/ns/iecUniTest/fc/assertEqual_LREAL.md *)
    VAR_INPUT
        act : LREAL; (*Variable to test*)
        xp : LREAL; (*Variable to test against*)
    END_VAR
END_FUNCTION
FUNCTION assertEqual_STRING : BOOL (* Returns TRUE if act = xp. *)(* https://github.com/tkucic/iecUniTest/blob/main/docs/docs/ns/iecUniTest/fc/assertEqual_STRING.md *)
    VAR_INPUT
        act : STRING; (*Variable to test*)
        xp : STRING; (*Variable to test against*)
    END_VAR
END_FUNCTION
FUNCTION assertEqual_WSTRING : BOOL (* Returns TRUE if act = xp. *)(* https://github.com/tkucic/iecUniTest/blob/main/docs/docs/ns/iecUniTest/fc/assertEqual_WSTRING.md *)
    VAR_INPUT
        act : WSTRING; (*Variable to test*)
        xp : WSTRING; (*Variable to test against*)
    END_VAR
END_FUNCTION
FUNCTION assertEqual_TIME : BOOL (* Returns TRUE if act = xp. *)(* https://github.com/tkucic/iecUniTest/blob/main/docs/docs/ns/iecUniTest/fc/assertEqual_TIME.md *)
    VAR_INPUT
        act : TIME; (*Variable to test*)
        xp : TIME; (*Variable to test against*)
    END_VAR
END_FUNCTION
FUNCTION assertEqual_DATE : BOOL (* Returns TRUE if act = xp. *)(* https://github.com/tkucic/iecUniTest/blob/main/docs/docs/ns/iecUniTest/fc/assertEqual_DATE.md *)
    VAR_INPUT
        act : DATE; (*Variable to test*)
        xp : DATE; (*Variable to test against*)
    END_VAR
END_FUNCTION
FUNCTION assertEqual_DATE_AND_TIME : BOOL (* Returns TRUE if act = xp. *)(* https://github.com/tkucic/iecUniTest/blob/main/docs/docs/ns/iecUniTest/fc/assertEqual_DATE_AND_TIME.md *)
    VAR_INPUT
        act : DT; (*Variable to test*)
        xp : DT; (*Variable to test against*)
    END_VAR
END_FUNCTION
FUNCTION assertEqual_TIME_OF_DAY : BOOL (* Returns TRUE if act = xp. *)(* https://github.com/tkucic/iecUniTest/blob/main/docs/docs/ns/iecUniTest/fc/assertEqual_TIME_OF_DAY.md *)
    VAR_INPUT
        act : TOD; (*Variable to test*)
        xp : TOD; (*Variable to test against*)
    END_VAR
END_FUNCTION
FUNCTION assertNotEqual_BOOL : BOOL (* Returns TRUE if act <> xp. *)(* https://github.com/tkucic/iecUniTest/blob/main/docs/docs/ns/iecUniTest/fc/assertNotEqual_BOOL.md *)
    VAR_INPUT
        act : BOOL; (*Variable to test*)
        xp : BOOL; (*Variable to test against*)
    END_VAR
END_FUNCTION
FUNCTION assertNotEqual_BYTE : BOOL (* Returns TRUE if act <> xp. *)(* https://github.com/tkucic/iecUniTest/blob/main/docs/docs/ns/iecUniTest/fc/assertNotEqual_BYTE.md *)
    VAR_INPUT
        act : BYTE; (*Variable to test*)
        xp : BYTE; (*Variable to test against*)
    END_VAR
END_FUNCTION
FUNCTION assertNotEqual_WORD : BOOL (* Returns TRUE if act <> xp. *)(* https://github.com/tkucic/iecUniTest/blob/main/docs/docs/ns/iecUniTest/fc/assertNotEqual_WORD.md *)
    VAR_INPUT
        act : WORD; (*Variable to test*)
        xp : WORD; (*Variable to test against*)
    END_VAR
END_FUNCTION
FUNCTION assertNotEqual_DWORD : BOOL (* Returns TRUE if act <> xp. *)(* https://github.com/tkucic/iecUniTest/blob/main/docs/docs/ns/iecUniTest/fc/assertNotEqual_DWORD.md *)
    VAR_INPUT
        act : DWORD; (*Variable to test*)
        xp : DWORD; (*Variable to test against*)
    END_VAR
END_FUNCTION
FUNCTION assertNotEqual_SINT : BOOL (* Returns TRUE if act <> xp. *)(* https://github.com/tkucic/iecUniTest/blob/main/docs/docs/ns/iecUniTest/fc/assertNotEqual_SINT.md *)
    VAR_INPUT
        act : SINT; (*Variable to test*)
        xp : SINT; (*Variable to test against*)
    END_VAR
END_FUNCTION
FUNCTION assertNotEqual_USINT : BOOL (* Returns TRUE if act <> xp. *)(* https://github.com/tkucic/iecUniTest/blob/main/docs/docs/ns/iecUniTest/fc/assertNotEqual_USINT.md *)
    VAR_INPUT
        act : USINT; (*Variable to test*)
        xp : USINT; (*Variable to test against*)
    END_VAR
END_FUNCTION
FUNCTION assertNotEqual_INT : BOOL (* Returns TRUE if act <> xp. *)(* https://github.com/tkucic/iecUniTest/blob/main/docs/docs/ns/iecUniTest/fc/assertNotEqual_INT.md *)
    VAR_INPUT
        act : INT; (*Variable to test*)
        xp : INT; (*Variable to test against*)
    END_VAR
END_FUNCTION
FUNCTION assertNotEqual_UINT : BOOL (* Returns TRUE if act <> xp. *)(* https://github.com/tkucic/iecUniTest/blob/main/docs/docs/ns/iecUniTest/fc/assertNotEqual_UINT.md *)
    VAR_INPUT
        act : UINT; (*Variable to test*)
        xp : UINT; (*Variable to test against*)
    END_VAR
END_FUNCTION
FUNCTION assertNotEqual_DINT : BOOL (* Returns TRUE if act <> xp. *)(* https://github.com/tkucic/iecUniTest/blob/main/docs/docs/ns/iecUniTest/fc/assertNotEqual_DINT.md *)
    VAR_INPUT
        act : DINT; (*Variable to test*)
        xp : DINT; (*Variable to test against*)
    END_VAR
END_FUNCTION
FUNCTION assertNotEqual_UDINT : BOOL (* Returns TRUE if act <> xp. *)(* https://github.com/tkucic/iecUniTest/blob/main/docs/docs/ns/iecUniTest/fc/assertNotEqual_UDINT.md *)
    VAR_INPUT
        act : UDINT; (*Variable to test*)
        xp : UDINT; (*Variable to test against*)
    END_VAR
END_FUNCTION
FUNCTION assertNotEqual_REAL : BOOL (* Returns TRUE if act <> xp. *)(* https://github.com/tkucic/iecUniTest/blob/main/docs/docs/ns/iecUniTest/fc/assertNotEqual_REAL.md *)
    VAR_INPUT
        act : REAL; (*Variable to test*)
        xp : REAL; (*Variable to test against*)
    END_VAR
END_FUNCTION
FUNCTION assertNotEqual_LREAL : BOOL (* Returns TRUE if act <> xp. *)(* https://github.com/tkucic/iecUniTest/blob/main/docs/docs/ns/iecUniTest/fc/assertNotEqual_LREAL.md *)
    VAR_INPUT
        act : LREAL; (*Variable to test*)
        xp : LREAL; (*Variable to test against*)
    END_VAR
END_FUNCTION
FUNCTION assertNotEqual_STRING : BOOL (* Returns TRUE if act <> xp. *)(* https://github.com/tkucic/iecUniTest/blob/main/docs/docs/ns/iecUniTest/fc/assertNotEqual_STRING.md *)
    VAR_INPUT
        act : STRING; (*Variable to test*)
        xp : STRING; (*Variable to test against*)
    END_VAR
END_FUNCTION
FUNCTION assertNotEqual_WSTRING : BOOL (* Returns TRUE if act <> xp. *)(* https://github.com/tkucic/iecUniTest/blob/main/docs/docs/ns/iecUniTest/fc/assertNotEqual_WSTRING.md *)
    VAR_INPUT
        act : WSTRING; (*Variable to test*)
        xp : WSTRING; (*Variable to test against*)
    END_VAR
END_FUNCTION
FUNCTION assertNotEqual_TIME : BOOL (* Returns TRUE if act <> xp. *)(* https://github.com/tkucic/iecUniTest/blob/main/docs/docs/ns/iecUniTest/fc/assertNotEqual_TIME.md *)
    VAR_INPUT
        act : TIME; (*Variable to test*)
        xp : TIME; (*Variable to test against*)
    END_VAR
END_FUNCTION
FUNCTION assertNotEqual_DATE : BOOL (* Returns TRUE if act <> xp. *)(* https://github.com/tkucic/iecUniTest/blob/main/docs/docs/ns/iecUniTest/fc/assertNotEqual_DATE.md *)
    VAR_INPUT
        act : DATE; (*Variable to test*)
        xp : DATE; (*Variable to test against*)
    END_VAR
END_FUNCTION
FUNCTION assertNotEqual_DATE_AND_TIME : BOOL (* Returns TRUE if act <> xp. *)(* https://github.com/tkucic/iecUniTest/blob/main/docs/docs/ns/iecUniTest/fc/assertNotEqual_DATE_AND_TIME.md *)
    VAR_INPUT
        act : DT; (*Variable to test*)
        xp : DT; (*Variable to test against*)
    END_VAR
END_FUNCTION
FUNCTION assertNotEqual_TIME_OF_DAY : BOOL (* Returns TRUE if act <> xp. *)(* https://github.com/tkucic/iecUniTest/blob/main/docs/docs/ns/iecUniTest/fc/assertNotEqual_TIME_OF_DAY.md *)
    VAR_INPUT
        act : TOD; (*Variable to test*)
        xp : TOD; (*Variable to test against*)
    END_VAR
END_FUNCTION
FUNCTION assertGreater_BYTE : BOOL (* Returns TRUE if act > xp. *)(* https://github.com/tkucic/iecUniTest/blob/main/docs/docs/ns/iecUniTest/fc/assertGreater_BYTE.md *)
    VAR_INPUT
        act : BYTE; (*Variable to test*)
        xp : BYTE; (*Variable to test against*)
    END_VAR
END_FUNCTION
FUNCTION assertGreater_WORD : BOOL (* Returns TRUE if act > xp. *)(* https://github.com/tkucic/iecUniTest/blob/main/docs/docs/ns/iecUniTest/fc/assertGreater_WORD.md *)
    VAR_INPUT
        act : WORD; (*Variable to test*)
        xp : WORD; (*Variable to test against*)
    END_VAR
END_FUNCTION
FUNCTION assertGreater_DWORD : BOOL (* Returns TRUE if act > xp. *)(* https://github.com/tkucic/iecUniTest/blob/main/docs/docs/ns/iecUniTest/fc/assertGreater_DWORD.md *)
    VAR_INPUT
        act : DWORD; (*Variable to test*)
        xp : DWORD; (*Variable to test against*)
    END_VAR
END_FUNCTION
FUNCTION assertGreater_SINT : BOOL (* Returns TRUE if act > xp. *)(* https://github.com/tkucic/iecUniTest/blob/main/docs/docs/ns/iecUniTest/fc/assertGreater_SINT.md *)
    VAR_INPUT
        act : SINT; (*Variable to test*)
        xp : SINT; (*Variable to test against*)
    END_VAR
END_FUNCTION
FUNCTION assertGreater_USINT : BOOL (* Returns TRUE if act > xp. *)(* https://github.com/tkucic/iecUniTest/blob/main/docs/docs/ns/iecUniTest/fc/assertGreater_USINT.md *)
    VAR_INPUT
        act : USINT; (*Variable to test*)
        xp : USINT; (*Variable to test against*)
    END_VAR
END_FUNCTION
FUNCTION assertGreater_INT : BOOL (* Returns TRUE if act > xp. *)(* https://github.com/tkucic/iecUniTest/blob/main/docs/docs/ns/iecUniTest/fc/assertGreater_INT.md *)
    VAR_INPUT
        act : INT; (*Variable to test*)
        xp : INT; (*Variable to test against*)
    END_VAR
END_FUNCTION
FUNCTION assertGreater_UINT : BOOL (* Returns TRUE if act > xp. *)(* https://github.com/tkucic/iecUniTest/blob/main/docs/docs/ns/iecUniTest/fc/assertGreater_UINT.md *)
    VAR_INPUT
        act : UINT; (*Variable to test*)
        xp : UINT; (*Variable to test against*)
    END_VAR
END_FUNCTION
FUNCTION assertGreater_DINT : BOOL (* Returns TRUE if act > xp. *)(* https://github.com/tkucic/iecUniTest/blob/main/docs/docs/ns/iecUniTest/fc/assertGreater_DINT.md *)
    VAR_INPUT
        act : DINT; (*Variable to test*)
        xp : DINT; (*Variable to test against*)
    END_VAR
END_FUNCTION
FUNCTION assertGreater_UDINT : BOOL (* Returns TRUE if act > xp. *)(* https://github.com/tkucic/iecUniTest/blob/main/docs/docs/ns/iecUniTest/fc/assertGreater_UDINT.md *)
    VAR_INPUT
        act : UDINT; (*Variable to test*)
        xp : UDINT; (*Variable to test against*)
    END_VAR
END_FUNCTION
FUNCTION assertGreater_REAL : BOOL (* Returns TRUE if act > xp. *)(* https://github.com/tkucic/iecUniTest/blob/main/docs/docs/ns/iecUniTest/fc/assertGreater_REAL.md *)
    VAR_INPUT
        act : REAL; (*Variable to test*)
        xp : REAL; (*Variable to test against*)
    END_VAR
END_FUNCTION
FUNCTION assertGreater_LREAL : BOOL (* Returns TRUE if act > xp. *)(* https://github.com/tkucic/iecUniTest/blob/main/docs/docs/ns/iecUniTest/fc/assertGreater_LREAL.md *)
    VAR_INPUT
        act : LREAL; (*Variable to test*)
        xp : LREAL; (*Variable to test against*)
    END_VAR
END_FUNCTION
FUNCTION assertGreater_TIME : BOOL (* Returns TRUE if act > xp. *)(* https://github.com/tkucic/iecUniTest/blob/main/docs/docs/ns/iecUniTest/fc/assertGreater_TIME.md *)
    VAR_INPUT
        act : TIME; (*Variable to test*)
        xp : TIME; (*Variable to test against*)
    END_VAR
END_FUNCTION
FUNCTION assertGreater_DATE : BOOL (* Returns TRUE if act > xp. *)(* https://github.com/tkucic/iecUniTest/blob/main/docs/docs/ns/iecUniTest/fc/assertGreater_DATE.md *)
    VAR_INPUT
        act : DATE; (*Variable to test*)
        xp : DATE; (*Variable to test against*)
    END_VAR
END_FUNCTION
FUNCTION assertGreater_DATE_AND_TIME : BOOL (* Returns TRUE if act > xp. *)(* https://github.com/tkucic/iecUniTest/blob/main/docs/docs/ns/iecUniTest/fc/assertGreater_DATE_AND_TIME.md *)
    VAR_INPUT
        act : DT; (*Variable to test*)
        xp : DT; (*Variable to test against*)
    END_VAR
END_FUNCTION
FUNCTION assertGreater_TIME_OF_DAY : BOOL (* Returns TRUE if act > xp. *)(* https://github.com/tkucic/iecUniTest/blob/main/docs/docs/ns/iecUniTest/fc/assertGreater_TIME_OF_DAY.md *)
    VAR_INPUT
        act : TOD; (*Variable to test*)
        xp : TOD; (*Variable to test against*)
    END_VAR
END_FUNCTION
FUNCTION assertGreaterEqual_BYTE : BOOL (* Returns TRUE if act >= xp. *)(* https://github.com/tkucic/iecUniTest/blob/main/docs/docs/ns/iecUniTest/fc/assertGreaterEqual_BYTE.md *)
    VAR_INPUT
        act : BYTE; (*Variable to test*)
        xp : BYTE; (*Variable to test against*)
    END_VAR
END_FUNCTION
FUNCTION assertGreaterEqual_WORD : BOOL (* Returns TRUE if act >= xp. *)(* https://github.com/tkucic/iecUniTest/blob/main/docs/docs/ns/iecUniTest/fc/assertGreaterEqual_WORD.md *)
    VAR_INPUT
        act : WORD; (*Variable to test*)
        xp : WORD; (*Variable to test against*)
    END_VAR
END_FUNCTION
FUNCTION assertGreaterEqual_DWORD : BOOL (* Returns TRUE if act >= xp. *)(* https://github.com/tkucic/iecUniTest/blob/main/docs/docs/ns/iecUniTest/fc/assertGreaterEqual_DWORD.md *)
    VAR_INPUT
        act : DWORD; (*Variable to test*)
        xp : DWORD; (*Variable to test against*)
    END_VAR
END_FUNCTION
FUNCTION assertGreaterEqual_SINT : BOOL (* Returns TRUE if act >= xp. *)(* https://github.com/tkucic/iecUniTest/blob/main/docs/docs/ns/iecUniTest/fc/assertGreaterEqual_SINT.md *)
    VAR_INPUT
        act : SINT; (*Variable to test*)
        xp : SINT; (*Variable to test against*)
    END_VAR
END_FUNCTION
FUNCTION assertGreaterEqual_USINT : BOOL (* Returns TRUE if act >= xp. *)(* https://github.com/tkucic/iecUniTest/blob/main/docs/docs/ns/iecUniTest/fc/assertGreaterEqual_USINT.md *)
    VAR_INPUT
        act : USINT; (*Variable to test*)
        xp : USINT; (*Variable to test against*)
    END_VAR
END_FUNCTION
FUNCTION assertGreaterEqual_INT : BOOL (* Returns TRUE if act >= xp. *)(* https://github.com/tkucic/iecUniTest/blob/main/docs/docs/ns/iecUniTest/fc/assertGreaterEqual_INT.md *)
    VAR_INPUT
        act : INT; (*Variable to test*)
        xp : INT; (*Variable to test against*)
    END_VAR
END_FUNCTION
FUNCTION assertGreaterEqual_UINT : BOOL (* Returns TRUE if act >= xp. *)(* https://github.com/tkucic/iecUniTest/blob/main/docs/docs/ns/iecUniTest/fc/assertGreaterEqual_UINT.md *)
    VAR_INPUT
        act : UINT; (*Variable to test*)
        xp : UINT; (*Variable to test against*)
    END_VAR
END_FUNCTION
FUNCTION assertGreaterEqual_DINT : BOOL (* Returns TRUE if act >= xp. *)(* https://github.com/tkucic/iecUniTest/blob/main/docs/docs/ns/iecUniTest/fc/assertGreaterEqual_DINT.md *)
    VAR_INPUT
        act : DINT; (*Variable to test*)
        xp : DINT; (*Variable to test against*)
    END_VAR
END_FUNCTION
FUNCTION assertGreaterEqual_UDINT : BOOL (* Returns TRUE if act >= xp. *)(* https://github.com/tkucic/iecUniTest/blob/main/docs/docs/ns/iecUniTest/fc/assertGreaterEqual_UDINT.md *)
    VAR_INPUT
        act : UDINT; (*Variable to test*)
        xp : UDINT; (*Variable to test against*)
    END_VAR
END_FUNCTION
FUNCTION assertGreaterEqual_REAL : BOOL (* Returns TRUE if act >= xp. *)(* https://github.com/tkucic/iecUniTest/blob/main/docs/docs/ns/iecUniTest/fc/assertGreaterEqual_REAL.md *)
    VAR_INPUT
        act : REAL; (*Variable to test*)
        xp : REAL; (*Variable to test against*)
    END_VAR
END_FUNCTION
FUNCTION assertGreaterEqual_LREAL : BOOL (* Returns TRUE if act >= xp. *)(* https://github.com/tkucic/iecUniTest/blob/main/docs/docs/ns/iecUniTest/fc/assertGreaterEqual_LREAL.md *)
    VAR_INPUT
        act : LREAL; (*Variable to test*)
        xp : LREAL; (*Variable to test against*)
    END_VAR
END_FUNCTION
FUNCTION assertGreaterEqual_TIME : BOOL (* Returns TRUE if act >= xp. *)(* https://github.com/tkucic/iecUniTest/blob/main/docs/docs/ns/iecUniTest/fc/assertGreaterEqual_TIME.md *)
    VAR_INPUT
        act : TIME; (*Variable to test*)
        xp : TIME; (*Variable to test against*)
    END_VAR
END_FUNCTION
FUNCTION assertGreaterEqual_DATE : BOOL (* Returns TRUE if act >= xp. *)(* https://github.com/tkucic/iecUniTest/blob/main/docs/docs/ns/iecUniTest/fc/assertGreaterEqual_DATE.md *)
    VAR_INPUT
        act : DATE; (*Variable to test*)
        xp : DATE; (*Variable to test against*)
    END_VAR
END_FUNCTION
FUNCTION assertGreaterEqual_DATE_AND_TIME : BOOL (* Returns TRUE if act >= xp. *)(* https://github.com/tkucic/iecUniTest/blob/main/docs/docs/ns/iecUniTest/fc/assertGreaterEqual_DATE_AND_TIME.md *)
    VAR_INPUT
        act : DT; (*Variable to test*)
        xp : DT; (*Variable to test against*)
    END_VAR
END_FUNCTION
FUNCTION assertGreaterEqual_TIME_OF_DAY : BOOL (* Returns TRUE if act >= xp. *)(* https://github.com/tkucic/iecUniTest/blob/main/docs/docs/ns/iecUniTest/fc/assertGreaterEqual_TIME_OF_DAY.md *)
    VAR_INPUT
        act : TOD; (*Variable to test*)
        xp : TOD; (*Variable to test against*)
    END_VAR
END_FUNCTION
FUNCTION assertLess_BYTE : BOOL (* Returns TRUE if act < xp. *)(* https://github.com/tkucic/iecUniTest/blob/main/docs/docs/ns/iecUniTest/fc/assertLess_BYTE.md *)
    VAR_INPUT
        act : BYTE; (*Variable to test*)
        xp : BYTE; (*Variable to test against*)
    END_VAR
END_FUNCTION
FUNCTION assertLess_WORD : BOOL (* Returns TRUE if act < xp. *)(* https://github.com/tkucic/iecUniTest/blob/main/docs/docs/ns/iecUniTest/fc/assertLess_WORD.md *)
    VAR_INPUT
        act : WORD; (*Variable to test*)
        xp : WORD; (*Variable to test against*)
    END_VAR
END_FUNCTION
FUNCTION assertLess_DWORD : BOOL (* Returns TRUE if act < xp. *)(* https://github.com/tkucic/iecUniTest/blob/main/docs/docs/ns/iecUniTest/fc/assertLess_DWORD.md *)
    VAR_INPUT
        act : DWORD; (*Variable to test*)
        xp : DWORD; (*Variable to test against*)
    END_VAR
END_FUNCTION
FUNCTION assertLess_SINT : BOOL (* Returns TRUE if act < xp. *)(* https://github.com/tkucic/iecUniTest/blob/main/docs/docs/ns/iecUniTest/fc/assertLess_SINT.md *)
    VAR_INPUT
        act : SINT; (*Variable to test*)
        xp : SINT; (*Variable to test against*)
    END_VAR
END_FUNCTION
FUNCTION assertLess_USINT : BOOL (* Returns TRUE if act < xp. *)(* https://github.com/tkucic/iecUniTest/blob/main/docs/docs/ns/iecUniTest/fc/assertLess_USINT.md *)
    VAR_INPUT
        act : USINT; (*Variable to test*)
        xp : USINT; (*Variable to test against*)
    END_VAR
END_FUNCTION
FUNCTION assertLess_INT : BOOL (* Returns TRUE if act < xp. *)(* https://github.com/tkucic/iecUniTest/blob/main/docs/docs/ns/iecUniTest/fc/assertLess_INT.md *)
    VAR_INPUT
        act : INT; (*Variable to test*)
        xp : INT; (*Variable to test against*)
    END_VAR
END_FUNCTION
FUNCTION assertLess_UINT : BOOL (* Returns TRUE if act < xp. *)(* https://github.com/tkucic/iecUniTest/blob/main/docs/docs/ns/iecUniTest/fc/assertLess_UINT.md *)
    VAR_INPUT
        act : UINT; (*Variable to test*)
        xp : UINT; (*Variable to test against*)
    END_VAR
END_FUNCTION
FUNCTION assertLess_DINT : BOOL (* Returns TRUE if act < xp. *)(* https://github.com/tkucic/iecUniTest/blob/main/docs/docs/ns/iecUniTest/fc/assertLess_DINT.md *)
    VAR_INPUT
        act : DINT; (*Variable to test*)
        xp : DINT; (*Variable to test against*)
    END_VAR
END_FUNCTION
FUNCTION assertLess_UDINT : BOOL (* Returns TRUE if act < xp. *)(* https://github.com/tkucic/iecUniTest/blob/main/docs/docs/ns/iecUniTest/fc/assertLess_UDINT.md *)
    VAR_INPUT
        act : UDINT; (*Variable to test*)
        xp : UDINT; (*Variable to test against*)
    END_VAR
END_FUNCTION
FUNCTION assertLess_REAL : BOOL (* Returns TRUE if act < xp. *)(* https://github.com/tkucic/iecUniTest/blob/main/docs/docs/ns/iecUniTest/fc/assertLess_REAL.md *)
    VAR_INPUT
        act : REAL; (*Variable to test*)
        xp : REAL; (*Variable to test against*)
    END_VAR
END_FUNCTION
FUNCTION assertLess_LREAL : BOOL (* Returns TRUE if act < xp. *)(* https://github.com/tkucic/iecUniTest/blob/main/docs/docs/ns/iecUniTest/fc/assertLess_LREAL.md *)
    VAR_INPUT
        act : LREAL; (*Variable to test*)
        xp : LREAL; (*Variable to test against*)
    END_VAR
END_FUNCTION
FUNCTION assertLess_TIME : BOOL (* Returns TRUE if act < xp. *)(* https://github.com/tkucic/iecUniTest/blob/main/docs/docs/ns/iecUniTest/fc/assertLess_TIME.md *)
    VAR_INPUT
        act : TIME; (*Variable to test*)
        xp : TIME; (*Variable to test against*)
    END_VAR
END_FUNCTION
FUNCTION assertLess_DATE : BOOL (* Returns TRUE if act < xp. *)(* https://github.com/tkucic/iecUniTest/blob/main/docs/docs/ns/iecUniTest/fc/assertLess_DATE.md *)
    VAR_INPUT
        act : DATE; (*Variable to test*)
        xp : DATE; (*Variable to test against*)
    END_VAR
END_FUNCTION
FUNCTION assertLess_DATE_AND_TIME : BOOL (* Returns TRUE if act < xp. *)(* https://github.com/tkucic/iecUniTest/blob/main/docs/docs/ns/iecUniTest/fc/assertLess_DATE_AND_TIME.md *)
    VAR_INPUT
        act : DT; (*Variable to test*)
        xp : DT; (*Variable to test against*)
    END_VAR
END_FUNCTION
FUNCTION assertLess_TIME_OF_DAY : BOOL (* Returns TRUE if act < xp. *)(* https://github.com/tkucic/iecUniTest/blob/main/docs/docs/ns/iecUniTest/fc/assertLess_TIME_OF_DAY.md *)
    VAR_INPUT
        act : TOD; (*Variable to test*)
        xp : TOD; (*Variable to test against*)
    END_VAR
END_FUNCTION
FUNCTION assertLessEqual_BYTE : BOOL (* Returns TRUE if act <= xp. *)(* https://github.com/tkucic/iecUniTest/blob/main/docs/docs/ns/iecUniTest/fc/assertLessEqual_BYTE.md *)
    VAR_INPUT
        act : BYTE; (*Variable to test*)
        xp : BYTE; (*Variable to test against*)
    END_VAR
END_FUNCTION
FUNCTION assertLessEqual_WORD : BOOL (* Returns TRUE if act <= xp. *)(* https://github.com/tkucic/iecUniTest/blob/main/docs/docs/ns/iecUniTest/fc/assertLessEqual_WORD.md *)
    VAR_INPUT
        act : WORD; (*Variable to test*)
        xp : WORD; (*Variable to test against*)
    END_VAR
END_FUNCTION
FUNCTION assertLessEqual_DWORD : BOOL (* Returns TRUE if act <= xp. *)(* https://github.com/tkucic/iecUniTest/blob/main/docs/docs/ns/iecUniTest/fc/assertLessEqual_DWORD.md *)
    VAR_INPUT
        act : DWORD; (*Variable to test*)
        xp : DWORD; (*Variable to test against*)
    END_VAR
END_FUNCTION
FUNCTION assertLessEqual_SINT : BOOL (* Returns TRUE if act <= xp. *)(* https://github.com/tkucic/iecUniTest/blob/main/docs/docs/ns/iecUniTest/fc/assertLessEqual_SINT.md *)
    VAR_INPUT
        act : SINT; (*Variable to test*)
        xp : SINT; (*Variable to test against*)
    END_VAR
END_FUNCTION
FUNCTION assertLessEqual_USINT : BOOL (* Returns TRUE if act <= xp. *)(* https://github.com/tkucic/iecUniTest/blob/main/docs/docs/ns/iecUniTest/fc/assertLessEqual_USINT.md *)
    VAR_INPUT
        act : USINT; (*Variable to test*)
        xp : USINT; (*Variable to test against*)
    END_VAR
END_FUNCTION
FUNCTION assertLessEqual_INT : BOOL (* Returns TRUE if act <= xp. *)(* https://github.com/tkucic/iecUniTest/blob/main/docs/docs/ns/iecUniTest/fc/assertLessEqual_INT.md *)
    VAR_INPUT
        act : INT; (*Variable to test*)
        xp : INT; (*Variable to test against*)
    END_VAR
END_FUNCTION
FUNCTION assertLessEqual_UINT : BOOL (* Returns TRUE if act <= xp. *)(* https://github.com/tkucic/iecUniTest/blob/main/docs/docs/ns/iecUniTest/fc/assertLessEqual_UINT.md *)
    VAR_INPUT
        act : UINT; (*Variable to test*)
        xp : UINT; (*Variable to test against*)
    END_VAR
END_FUNCTION
FUNCTION assertLessEqual_DINT : BOOL (* Returns TRUE if act <= xp. *)(* https://github.com/tkucic/iecUniTest/blob/main/docs/docs/ns/iecUniTest/fc/assertLessEqual_DINT.md *)
    VAR_INPUT
        act : DINT; (*Variable to test*)
        xp : DINT; (*Variable to test against*)
    END_VAR
END_FUNCTION
FUNCTION assertLessEqual_UDINT : BOOL (* Returns TRUE if act <= xp. *)(* https://github.com/tkucic/iecUniTest/blob/main/docs/docs/ns/iecUniTest/fc/assertLessEqual_UDINT.md *)
    VAR_INPUT
        act : UDINT; (*Variable to test*)
        xp : UDINT; (*Variable to test against*)
    END_VAR
END_FUNCTION
FUNCTION assertLessEqual_REAL : BOOL (* Returns TRUE if act <= xp. *)(* https://github.com/tkucic/iecUniTest/blob/main/docs/docs/ns/iecUniTest/fc/assertLessEqual_REAL.md *)
    VAR_INPUT
        act : REAL; (*Variable to test*)
        xp : REAL; (*Variable to test against*)
    END_VAR
END_FUNCTION
FUNCTION assertLessEqual_LREAL : BOOL (* Returns TRUE if act <= xp. *)(* https://github.com/tkucic/iecUniTest/blob/main/docs/docs/ns/iecUniTest/fc/assertLessEqual_LREAL.md *)
    VAR_INPUT
        act : LREAL; (*Variable to test*)
        xp : LREAL; (*Variable to test against*)
    END_VAR
END_FUNCTION
FUNCTION assertLessEqual_TIME : BOOL (* Returns TRUE if act <= xp. *)(* https://github.com/tkucic/iecUniTest/blob/main/docs/docs/ns/iecUniTest/fc/assertLessEqual_TIME.md *)
    VAR_INPUT
        act : TIME; (*Variable to test*)
        xp : TIME; (*Variable to test against*)
    END_VAR
END_FUNCTION
FUNCTION assertLessEqual_DATE : BOOL (* Returns TRUE if act <= xp. *)(* https://github.com/tkucic/iecUniTest/blob/main/docs/docs/ns/iecUniTest/fc/assertLessEqual_DATE.md *)
    VAR_INPUT
        act : DATE; (*Variable to test*)
        xp : DATE; (*Variable to test against*)
    END_VAR
END_FUNCTION
FUNCTION assertLessEqual_DATE_AND_TIME : BOOL (* Returns TRUE if act <= xp. *)(* https://github.com/tkucic/iecUniTest/blob/main/docs/docs/ns/iecUniTest/fc/assertLessEqual_DATE_AND_TIME.md *)
    VAR_INPUT
        act : DT; (*Variable to test*)
        xp : DT; (*Variable to test against*)
    END_VAR
END_FUNCTION
FUNCTION assertLessEqual_TIME_OF_DAY : BOOL (* Returns TRUE if act <= xp. *)(* https://github.com/tkucic/iecUniTest/blob/main/docs/docs/ns/iecUniTest/fc/assertLessEqual_TIME_OF_DAY.md *)
    VAR_INPUT
        act : TOD; (*Variable to test*)
        xp : TOD; (*Variable to test against*)
    END_VAR
END_FUNCTION
FUNCTION assertArrayEqual_BOOL : BOOL (* Returns TRUE if act == xp. *)(* https://github.com/tkucic/iecUniTest/blob/main/docs/docs/ns/iecUniTest/fc/assertArrayEqual_BOOL.md *)
    VAR_INPUT
        act : REFERENCE TO ARRAY[0..32000] OF BOOL; (*Variable to test*)
        xp : REFERENCE TO ARRAY[0..32000] OF BOOL; (*Variable to test against*)
        size : UINT; (*Size of the array (ADR(act))*)
    END_VAR
    VAR
        i : UINT; (*Iterator variable*)
        vStop : UINT; (*Size of the array / End of iteration*)
        pt1 : REFERENCE TO BOOL; (*Pointer to the element of the array act*)
        pt2 : REFERENCE TO BOOL; (*Pointer to the element of the array xp*)
    END_VAR
END_FUNCTION
FUNCTION assertArrayEqual_BYTE : BOOL (* Returns TRUE if act == xp. *)(* https://github.com/tkucic/iecUniTest/blob/main/docs/docs/ns/iecUniTest/fc/assertArrayEqual_BYTE.md *)
    VAR_INPUT
        act : REFERENCE TO ARRAY[0..32000] OF BYTE; (*Variable to test*)
        xp : REFERENCE TO ARRAY[0..32000] OF BYTE; (*Variable to test against*)
        size : UINT; (*Size of the array (ADR(act))*)
    END_VAR
    VAR
        i : UINT; (*Iterator variable*)
        vStop : UINT; (*Size of the array / End of iteration*)
        pt1 : REFERENCE TO BYTE; (*Pointer to the element of the array act*)
        pt2 : REFERENCE TO BYTE; (*Pointer to the element of the array xp*)
    END_VAR
END_FUNCTION
FUNCTION assertArrayEqual_WORD : BOOL (* Returns TRUE if act == xp. *)(* https://github.com/tkucic/iecUniTest/blob/main/docs/docs/ns/iecUniTest/fc/assertArrayEqual_WORD.md *)
    VAR_INPUT
        act : REFERENCE TO ARRAY[0..32000] OF WORD; (*Variable to test*)
        xp : REFERENCE TO ARRAY[0..32000] OF WORD; (*Variable to test against*)
        size : UINT; (*Size of the array (ADR(act))*)
    END_VAR
    VAR
        i : UINT; (*Iterator variable*)
        vStop : UINT; (*Size of the array / End of iteration*)
        pt1 : REFERENCE TO WORD; (*Pointer to the element of the array act*)
        pt2 : REFERENCE TO WORD; (*Pointer to the element of the array xp*)
    END_VAR
END_FUNCTION
FUNCTION assertArrayEqual_DWORD : BOOL (* Returns TRUE if act == xp. *)(* https://github.com/tkucic/iecUniTest/blob/main/docs/docs/ns/iecUniTest/fc/assertArrayEqual_DWORD.md *)
    VAR_INPUT
        act : REFERENCE TO ARRAY[0..32000] OF DWORD; (*Variable to test*)
        xp : REFERENCE TO ARRAY[0..32000] OF DWORD; (*Variable to test against*)
        size : UINT; (*Size of the array (ADR(act))*)
    END_VAR
    VAR
        i : UINT; (*Iterator variable*)
        vStop : UINT; (*Size of the array / End of iteration*)
        pt1 : REFERENCE TO DWORD; (*Pointer to the element of the array act*)
        pt2 : REFERENCE TO DWORD; (*Pointer to the element of the array xp*)
    END_VAR
END_FUNCTION
FUNCTION assertArrayEqual_SINT : BOOL (* Returns TRUE if act == xp. *)(* https://github.com/tkucic/iecUniTest/blob/main/docs/docs/ns/iecUniTest/fc/assertArrayEqual_SINT.md *)
    VAR_INPUT
        act : REFERENCE TO ARRAY[0..32000] OF SINT; (*Variable to test*)
        xp : REFERENCE TO ARRAY[0..32000] OF SINT; (*Variable to test against*)
        size : UINT; (*Size of the array (ADR(act))*)
    END_VAR
    VAR
        i : UINT; (*Iterator variable*)
        vStop : UINT; (*Size of the array / End of iteration*)
        pt1 : REFERENCE TO SINT; (*Pointer to the element of the array act*)
        pt2 : REFERENCE TO SINT; (*Pointer to the element of the array xp*)
    END_VAR
END_FUNCTION
FUNCTION assertArrayEqual_USINT : BOOL (* Returns TRUE if act == xp. *)(* https://github.com/tkucic/iecUniTest/blob/main/docs/docs/ns/iecUniTest/fc/assertArrayEqual_USINT.md *)
    VAR_INPUT
        act : REFERENCE TO ARRAY[0..32000] OF USINT; (*Variable to test*)
        xp : REFERENCE TO ARRAY[0..32000] OF USINT; (*Variable to test against*)
        size : UINT; (*Size of the array (ADR(act))*)
    END_VAR
    VAR
        i : UINT; (*Iterator variable*)
        vStop : UINT; (*Size of the array / End of iteration*)
        pt1 : REFERENCE TO USINT; (*Pointer to the element of the array act*)
        pt2 : REFERENCE TO USINT; (*Pointer to the element of the array xp*)
    END_VAR
END_FUNCTION
FUNCTION assertArrayEqual_INT : BOOL (* Returns TRUE if act == xp. *)(* https://github.com/tkucic/iecUniTest/blob/main/docs/docs/ns/iecUniTest/fc/assertArrayEqual_INT.md *)
    VAR_INPUT
        act : REFERENCE TO ARRAY[0..32000] OF INT; (*Variable to test*)
        xp : REFERENCE TO ARRAY[0..32000] OF INT; (*Variable to test against*)
        size : UINT; (*Size of the array (ADR(act))*)
    END_VAR
    VAR
        i : UINT; (*Iterator variable*)
        vStop : UINT; (*Size of the array / End of iteration*)
        pt1 : REFERENCE TO INT; (*Pointer to the element of the array act*)
        pt2 : REFERENCE TO INT; (*Pointer to the element of the array xp*)
    END_VAR
END_FUNCTION
FUNCTION assertArrayEqual_UINT : BOOL (* Returns TRUE if act == xp. *)(* https://github.com/tkucic/iecUniTest/blob/main/docs/docs/ns/iecUniTest/fc/assertArrayEqual_UINT.md *)
    VAR_INPUT
        act : REFERENCE TO ARRAY[0..32000] OF UINT; (*Variable to test*)
        xp : REFERENCE TO ARRAY[0..32000] OF UINT; (*Variable to test against*)
        size : UINT; (*Size of the array (ADR(act))*)
    END_VAR
    VAR
        i : UINT; (*Iterator variable*)
        vStop : UINT; (*Size of the array / End of iteration*)
        pt1 : REFERENCE TO UINT; (*Pointer to the element of the array act*)
        pt2 : REFERENCE TO UINT; (*Pointer to the element of the array xp*)
    END_VAR
END_FUNCTION
FUNCTION assertArrayEqual_DINT : BOOL (* Returns TRUE if act == xp. *)(* https://github.com/tkucic/iecUniTest/blob/main/docs/docs/ns/iecUniTest/fc/assertArrayEqual_DINT.md *)
    VAR_INPUT
        act : REFERENCE TO ARRAY[0..32000] OF DINT; (*Variable to test*)
        xp : REFERENCE TO ARRAY[0..32000] OF DINT; (*Variable to test against*)
        size : UINT; (*Size of the array (ADR(act))*)
    END_VAR
    VAR
        i : UINT; (*Iterator variable*)
        vStop : UINT; (*Size of the array / End of iteration*)
        pt1 : REFERENCE TO DINT; (*Pointer to the element of the array act*)
        pt2 : REFERENCE TO DINT; (*Pointer to the element of the array xp*)
    END_VAR
END_FUNCTION
FUNCTION assertArrayEqual_UDINT : BOOL (* Returns TRUE if act == xp. *)(* https://github.com/tkucic/iecUniTest/blob/main/docs/docs/ns/iecUniTest/fc/assertArrayEqual_UDINT.md *)
    VAR_INPUT
        act : REFERENCE TO ARRAY[0..32000] OF UDINT; (*Variable to test*)
        xp : REFERENCE TO ARRAY[0..32000] OF UDINT; (*Variable to test against*)
        size : UINT; (*Size of the array (ADR(act))*)
    END_VAR
    VAR
        i : UINT; (*Iterator variable*)
        vStop : UINT; (*Size of the array / End of iteration*)
        pt1 : REFERENCE TO UDINT; (*Pointer to the element of the array act*)
        pt2 : REFERENCE TO UDINT; (*Pointer to the element of the array xp*)
    END_VAR
END_FUNCTION
FUNCTION assertArrayEqual_REAL : BOOL (* Returns TRUE if act == xp. *)(* https://github.com/tkucic/iecUniTest/blob/main/docs/docs/ns/iecUniTest/fc/assertArrayEqual_REAL.md *)
    VAR_INPUT
        act : REFERENCE TO ARRAY[0..32000] OF REAL; (*Variable to test*)
        xp : REFERENCE TO ARRAY[0..32000] OF REAL; (*Variable to test against*)
        size : UINT; (*Size of the array (ADR(act))*)
    END_VAR
    VAR
        i : UINT; (*Iterator variable*)
        vStop : UINT; (*Size of the array / End of iteration*)
        pt1 : REFERENCE TO REAL; (*Pointer to the element of the array act*)
        pt2 : REFERENCE TO REAL; (*Pointer to the element of the array xp*)
    END_VAR
END_FUNCTION
FUNCTION assertArrayEqual_LREAL : BOOL (* Returns TRUE if act == xp. *)(* https://github.com/tkucic/iecUniTest/blob/main/docs/docs/ns/iecUniTest/fc/assertArrayEqual_LREAL.md *)
    VAR_INPUT
        act : REFERENCE TO ARRAY[0..32000] OF LREAL; (*Variable to test*)
        xp : REFERENCE TO ARRAY[0..32000] OF LREAL; (*Variable to test against*)
        size : UINT; (*Size of the array (ADR(act))*)
    END_VAR
    VAR
        i : UINT; (*Iterator variable*)
        vStop : UINT; (*Size of the array / End of iteration*)
        pt1 : REFERENCE TO LREAL; (*Pointer to the element of the array act*)
        pt2 : REFERENCE TO LREAL; (*Pointer to the element of the array xp*)
    END_VAR
END_FUNCTION
FUNCTION assertArrayEqual_STRING : BOOL (* Returns TRUE if act == xp. *)(* https://github.com/tkucic/iecUniTest/blob/main/docs/docs/ns/iecUniTest/fc/assertArrayEqual_STRING.md *)
    VAR_INPUT
        act : REFERENCE TO ARRAY[0..32000] OF STRING; (*Variable to test*)
        xp : REFERENCE TO ARRAY[0..32000] OF STRING; (*Variable to test against*)
        size : UINT; (*Size of the array (ADR(act))*)
    END_VAR
    VAR
        i : UINT; (*Iterator variable*)
        vStop : UINT; (*Size of the array / End of iteration*)
        pt1 : REFERENCE TO STRING; (*Pointer to the element of the array act*)
        pt2 : REFERENCE TO STRING; (*Pointer to the element of the array xp*)
    END_VAR
END_FUNCTION
FUNCTION assertArrayEqual_WSTRING : BOOL (* Returns TRUE if act == xp. *)(* https://github.com/tkucic/iecUniTest/blob/main/docs/docs/ns/iecUniTest/fc/assertArrayEqual_WSTRING.md *)
    VAR_INPUT
        act : REFERENCE TO ARRAY[0..32000] OF WSTRING; (*Variable to test*)
        xp : REFERENCE TO ARRAY[0..32000] OF WSTRING; (*Variable to test against*)
        size : UINT; (*Size of the array (ADR(act))*)
    END_VAR
    VAR
        i : UINT; (*Iterator variable*)
        vStop : UINT; (*Size of the array / End of iteration*)
        pt1 : REFERENCE TO WSTRING; (*Pointer to the element of the array act*)
        pt2 : REFERENCE TO WSTRING; (*Pointer to the element of the array xp*)
    END_VAR
END_FUNCTION
FUNCTION assertArrayEqual_TIME : BOOL (* Returns TRUE if act == xp. *)(* https://github.com/tkucic/iecUniTest/blob/main/docs/docs/ns/iecUniTest/fc/assertArrayEqual_TIME.md *)
    VAR_INPUT
        act : REFERENCE TO ARRAY[0..32000] OF TIME; (*Variable to test*)
        xp : REFERENCE TO ARRAY[0..32000] OF TIME; (*Variable to test against*)
        size : UINT; (*Size of the array (ADR(act))*)
    END_VAR
    VAR
        i : UINT; (*Iterator variable*)
        vStop : UINT; (*Size of the array / End of iteration*)
        pt1 : REFERENCE TO TIME; (*Pointer to the element of the array act*)
        pt2 : REFERENCE TO TIME; (*Pointer to the element of the array xp*)
    END_VAR
END_FUNCTION
FUNCTION assertArrayEqual_DATE : BOOL (* Returns TRUE if act == xp. *)(* https://github.com/tkucic/iecUniTest/blob/main/docs/docs/ns/iecUniTest/fc/assertArrayEqual_DATE.md *)
    VAR_INPUT
        act : REFERENCE TO ARRAY[0..32000] OF DATE; (*Variable to test*)
        xp : REFERENCE TO ARRAY[0..32000] OF DATE; (*Variable to test against*)
        size : UINT; (*Size of the array (ADR(act))*)
    END_VAR
    VAR
        i : UINT; (*Iterator variable*)
        vStop : UINT; (*Size of the array / End of iteration*)
        pt1 : REFERENCE TO DATE; (*Pointer to the element of the array act*)
        pt2 : REFERENCE TO DATE; (*Pointer to the element of the array xp*)
    END_VAR
END_FUNCTION
FUNCTION assertArrayEqual_DATE_AND_TIME : BOOL (* Returns TRUE if act == xp. *)(* https://github.com/tkucic/iecUniTest/blob/main/docs/docs/ns/iecUniTest/fc/assertArrayEqual_DATE_AND_TIME.md *)
    VAR_INPUT
        act : REFERENCE TO ARRAY[0..32000] OF DT; (*Variable to test*)
        xp : REFERENCE TO ARRAY[0..32000] OF DT; (*Variable to test against*)
        size : UINT; (*Size of the array (ADR(act))*)
    END_VAR
    VAR
        i : UINT; (*Iterator variable*)
        vStop : UINT; (*Size of the array / End of iteration*)
        pt1 : REFERENCE TO DT; (*Pointer to the element of the array act*)
        pt2 : REFERENCE TO DT; (*Pointer to the element of the array xp*)
    END_VAR
END_FUNCTION
FUNCTION assertArrayEqual_TIME_OF_DAY : BOOL (* Returns TRUE if act == xp. *)(* https://github.com/tkucic/iecUniTest/blob/main/docs/docs/ns/iecUniTest/fc/assertArrayEqual_TIME_OF_DAY.md *)
    VAR_INPUT
        act : REFERENCE TO ARRAY[0..32000] OF TOD; (*Variable to test*)
        xp : REFERENCE TO ARRAY[0..32000] OF TOD; (*Variable to test against*)
        size : UINT; (*Size of the array (ADR(act))*)
    END_VAR
    VAR
        i : UINT; (*Iterator variable*)
        vStop : UINT; (*Size of the array / End of iteration*)
        pt1 : REFERENCE TO TOD; (*Pointer to the element of the array act*)
        pt2 : REFERENCE TO TOD; (*Pointer to the element of the array xp*)
    END_VAR
END_FUNCTION
FUNCTION assertTrue : BOOL (* Returns TRUE if condition is TRUE *)(* https://github.com/tkucic/iecUniTest/blob/main/docs/docs/ns/iecUniTest/fc/assertTrue.md *)
    VAR_INPUT
        condition : BOOL; (*Variable to test*)
    END_VAR
END_FUNCTION
